	46: IF Laser_Marked THEN
			OP150_Laser_Start:=0;
			OP150b_Auto_Seq :=47;
		END_IF	
		
	47:	IF NOT OP150_Laser_Start AND Laser_Marked THEN
			OP150b_Auto_Seq :=50;
		ELSIF OP150_Laser_Failed THEN		//Laser_Mark_Delay.Q AND (OP150_Laser_Failed OR NOT OP150_Laser_Completed) THEN
			OP150_Laser_Start:=0;
			OP150b_Auto_Seq :=80;
		END_IF
		
	50: MOVER_CMP_STATUS[OP150B_LH_STN_MOVER][1]:=156;	
		OP150B_LH_STN_ENABLE:=0;
		IF MOVER_CMP_STATUS[OP150B_LH_STN_MOVER][1]=156 THEN
			STATION_DONE[OP150B_LH_STN_MOVER][OP150B_LH_XTS_POS_NO]			:= TRUE;
			OP150b_Auto_Seq :=30;
		END_IF		
	
	60: Rejection_Code:=Rejection_Codes_Function(Fixture_LH);
		OP150B_Text_OK:=0;
		OP150b_Auto_Seq :=61;
		
	61: Line_1						:= Rejection_Code;
		OP150_Lsr_String  			:= Line_1; 
		OP150_Lsr_Block_ID			:= 0;
		OP150_Lsr_Text_Change_Start := 1;
		OP150b_Auto_Seq :=62;
		
	62:IF OP150_Lsr_Text_Change_Complete THEN// NOT OP150_Lsr_Text_Change_Start THEN
			Txt_Changed:=0;
			OP150b_Auto_Seq :=66;
		END_IF	
		
	66:	OP150_Laser_Start := TRUE;
		IF OP150_Laser_Start THEN
			OP150b_Auto_Seq :=67;
		END_IF	
	
	67: IF Laser_Marked THEN
			OP150_Laser_Start:=0;
			OP150b_Auto_Seq :=68;
		END_IF	
		
	68: IF NOT OP150_Laser_Start AND Laser_Marked THEN
			OP150b_Auto_Seq :=69;
		ELSIF OP150_Laser_Failed THEN//Laser_Mark_Delay.Q AND (OP150_Laser_Failed OR NOT OP150_Laser_Completed) THEN
			OP150_Laser_Start:=0;
			OP150b_Auto_Seq :=80;
		END_IF	
		
	69: Job_Initialize:=1;
		IF OP150B_Text_OK THEN
			OP150b_Auto_Seq:=70;
		END_IF
		
	70: OP150B_LH_STN_ENABLE:=0;
		MOVER_CMP_STATUS[OP150B_LH_STN_MOVER][1]:=156;	
		IF MOVER_CMP_STATUS[OP150B_LH_STN_MOVER][1]=156 THEN
			STATION_DONE[OP150B_LH_STN_MOVER][OP150B_LH_XTS_POS_NO]			:= TRUE;
			OP150b_Auto_Seq :=30;
		END_IF	

    80: MOVER_CMP_STATUS[OP150B_LH_STN_MOVER][1]:=157;
		IF MOVER_CMP_STATUS[OP150B_LH_STN_MOVER][1]=157 THEN
			OP150B_LH_STN_ENABLE:=0;
			OP150B_RH_STN_ENABLE:=0;
			STATION_DONE[OP150B_LH_STN_MOVER][OP150B_LH_XTS_POS_NO]	:= TRUE;
			OP150b_Auto_Seq :=30;
		END_IF		
		
	100: IF OP150B_Text_OK THEN //NOT OP150_Lsr_Text_Change_Start THEN
			OP150_Laser_Start := TRUE;
			IF OP150_Laser_Start THEN
				OP150b_Auto_Seq :=106;
			END_IF	
		 END_IF	
		
	106:IF Laser_Marked THEN
			OP150_Laser_Start:=0;
			OP150b_Auto_Seq :=107;
		END_IF	
		
	107:IF NOT OP150_Laser_Start AND Laser_Marked THEN
			OP150b_Auto_Seq :=110;
		ELSIF OP150_Laser_Failed THEN//Laser_Mark_Delay.Q AND (OP150_Laser_Failed OR NOT OP150_Laser_Completed) THEN
			OP150_Laser_Start:=0;
			OP150b_Auto_Seq :=160;
		END_IF
		
	110: OP150B_RH_STN_ENABLE:=0;
		 MOVER_CMP_STATUS[OP150B_RH_STN_MOVER][2]:=156;	
		 IF MOVER_CMP_STATUS[OP150B_RH_STN_MOVER][2]=156 THEN
			STATION_DONE[OP150B_RH_STN_MOVER][OP150B_RH_XTS_POS_NO]			:= TRUE;
			OP150b_Auto_Seq :=30;
		 END_IF		

	140: Rejection_Code:=Rejection_Codes_Function(Fixture_RH);
		 OP150b_Auto_Seq :=141;
		
	141: Line_1						:= Rejection_Code;
		 OP150_Lsr_String  			:= Line_1; 
		 OP150_Lsr_Block_ID			:= 0;
		 OP150_Lsr_Text_Change_Start := 1;
		 OP150b_Auto_Seq :=142;
		 
	142: IF OP150_Lsr_Text_Change_Complete THEN //NOT OP150_Lsr_Text_Change_Start THEN			
			OP150b_Auto_Seq :=143;
		 END_IF	

	143:// Line_2			  			:= 'D7.89';
		 OP150_Lsr_String  			:= Line_2; 
		 OP150_Lsr_Block_ID			:= 65536;
		 OP150_Lsr_Text_Change_Start := 1;
		 OP150b_Auto_Seq :=144;
		 
	144: IF OP150_Lsr_Text_Change_Complete THEN // NOT OP150_Lsr_Text_Change_Start THEN
			OP150b_Auto_Seq :=145;
		 END_IF	
	 
	145: //Line_3			  			:='>PK25D<';
		 OP150_Lsr_String  			:= Line_3; 
		 OP150_Lsr_Block_ID			:= 131072;
		 OP150_Lsr_Text_Change_Start := 1;
		 OP150b_Auto_Seq :=146;
		 
	146: IF OP150_Lsr_Text_Change_Complete THEN // NOT OP150_Lsr_Text_Change_Start THEN
			OP150_Laser_Start := TRUE;
			IF OP150_Laser_Start THEN
				OP150b_Auto_Seq :=147;
			END_IF	
		 END_IF	
	
	147: OP150_Laser_Start:=0;
		IF NOT OP150_Laser_Start THEN
			OP150b_Auto_Seq :=148;
		END_IF		 
		 
	148: IF NOT OP150_Laser_Start AND Laser_Marked THEN
			OP150b_Auto_Seq :=150;
		 ELSIF Laser_Mark_Delay.Q AND OP150_Laser_Failed THEN // OR NOT OP150_Laser_Completed) THEN
			OP150_Laser_Start:=0;
			OP150b_Auto_Seq :=160;
		 END_IF	
		
	150: MOVER_CMP_STATUS[OP150B_RH_STN_MOVER][2]:=156;	
		 IF MOVER_CMP_STATUS[OP150B_RH_STN_MOVER][2]=156 THEN
			STATION_DONE[OP150B_RH_STN_MOVER][OP150B_RH_XTS_POS_NO]			:= TRUE;
			OP150B_RH_STN_ENABLE:=0;
			OP150b_Auto_Seq :=30;
		 END_IF	
		 
	160: OP150B_RH_STN_ENABLE:=0;
		 MOVER_CMP_STATUS[OP150B_RH_STN_MOVER][2]:=157;	
		 IF MOVER_CMP_STATUS[OP150B_RH_STN_MOVER][2]=157 THEN
			STATION_DONE[OP150B_RH_STN_MOVER][OP150B_RH_XTS_POS_NO]			:= TRUE;
			OP150b_Auto_Seq :=30;
		 END_IF		 
END_CASE

Laser_Mark_Delay(IN:= (OP150_HMI_Reset OR OP150_Laser_Start),PT:=T#1S);

IF Laser_Mark_Delay.Q THEN
	OP150_HMI_Reset:=0;
END_IF

//Timer(IN:=OP150b_Auto_Seq=46 OR OP150b_Auto_Seq=106 ,PT:=T#1500MS);
//Txt_Change_Tmr(IN:=OP150_Lsr_Text_Change_Start ,PT:=T#500MS);

//IF Txt_Change_Tmr.Q THEN
//	OP150_Lsr_Text_Change_Start:=0;
//END_IF

IF Dry_run THEN
	Fixture_LH	:=150;
	Fixture_RH  :=150;
ELSE	
   Fixture_LH:=MOVER_CMP_STATUS[OP150B_LH_STN_MOVER][1];
   Fixture_RH:=MOVER_CMP_STATUS[OP150B_RH_STN_MOVER][2];
END_IF


//***************************Job change according to model********************************************\\
IF OP150_Model='6.3' THEN
	OP150_Lsr_Job_ID:=131072;
ELSIF OP150_Model='7.89' THEN
	OP150_Lsr_Job_ID:=0;
END_IF

IF OP150_Model='6.3' AND OP150_Laser_FB.Curr_JOB_id=2 THEN
	OP150B_Job_OK:=1;
ELSIF OP150_Model='7.89' AND OP150_Laser_FB.Curr_JOB_id=0 THEN
	OP150B_Job_OK:=1;
ELSE
	OP150B_Job_OK:=0;
END_IF

CASE OP150b_Job_Change_Seq OF
	10: IF NOT OP150_B_ErrorActive THEN
		 	OP150b_Job_Change_Seq :=20;
		END_IF
		
	20: IF OP150_Lsr_Ready THEN
			OP150b_Job_Change_Seq :=30;
		END_IF
		
	25: IF OP150_Model='6.3' AND OP150_Laser_FB.Curr_JOB_id<>2 THEN
			OP150b_Job_Change_Seq :=30;
		ELSIF OP150_Model='7.89' AND OP150_Laser_FB.Curr_JOB_id<>0 THEN
			OP150b_Job_Change_Seq :=30; 	
		END_IF
		
	30: IF OP150_Laser_FB.Curr_JOB_id <> OP150_Lsr_Job_ID THEN
			OP150b_Job_Change_Seq :=40;
		END_IF
		
	40: OP150_Lsr_Job_Change_Start:=1;
		OP150b_Job_Change_Seq :=50;
	 		
	50: IF OP150_Lsr_Job_Change_Complete AND NOT OP150_Lsr_Job_Change_Start THEN
			OP150_Lsr_Job_Change_Start := 0;
			OP150b_Job_Change_Seq :=25;
		END_IF
	
END_CASE

//************************************ Lines change According to Model & Batch ********************\\

Temp_String:=CONCAT(WORD_TO_STRING(fbTime.systemTime.wDay),'-');//WORD_TO_STRING(fbTime.systemTime.wMonth));
Laser_Line1:=CONCAT(Temp_String,'Jan');

IF Line_1<>Laser_Line1 THEN
	Job_Initialize:=1;
END_IF

CASE OP150b_Text_Change_Seq OF 
	
	10: IF NOT OP150_B_ErrorActive THEN
		 	OP150b_Text_Change_Seq :=20;
		END_IF
		
	20: IF OP150_Lsr_Ready THEN
			OP150b_Text_Change_Seq :=30;
		END_IF

	30: IF Batch_Change OR Job_Initialize THEN
			OP150B_Text_OK:=0;
			OP150b_Text_Change_Seq :=40;
		END_IF
	
 	40:	 Line_1						 := Laser_Line1;
		 OP150_Lsr_String  			 := Line_1; 
		 OP150_Lsr_Block_ID			 := 0;
		 OP150b_Text_Change_Seq 	 :=41;
		 
	41:  OP150_Lsr_Text_Change_Start := 1;
		  OP150b_Text_Change_Seq 	 :=50;
		 
	50: IF OP150_Lsr_Text_Change_Complete THEN //NOT OP150_Lsr_Text_Change_Start THEN
			Txt_Changed:=0;
			OP150b_Text_Change_Seq 	 :=60;
		 END_IF	
		
	60:	OP150_Lsr_String  			:= Line_2; 
		OP150_Lsr_Block_ID			:= 65536;
		OP150_Lsr_Text_Change_Start := 1;
		OP150b_Text_Change_Seq 	 :=70;
		
	70:IF OP150_Lsr_Text_Change_Complete THEN //NOT OP150_Lsr_Text_Change_Start THEN
			Txt_Changed:=0;
			OP150b_Text_Change_Seq 	 :=80;
		END_IF	
	 
	80:	OP150_Lsr_String  			:= Line_3; 
		OP150_Lsr_Block_ID			:= 131072;
		OP150_Lsr_Text_Change_Start := 1;
		OP150b_Text_Change_Seq 	 :=90;

	90: IF OP150_Lsr_Text_Change_Complete THEN //NOT OP150_Lsr_Text_Change_Start THEN
			Txt_Changed:=0;
			OP150b_Text_Change_Seq 	 :=100;
		END_IF		
		
  100:	OP150B_Text_OK  :=1;
  		Batch_Change    :=0;
		Job_Initialize  :=0;
		OP150b_Text_Change_Seq 	 :=10;
END_CASE


//############################		OP150B STATION ENABLE CONDITION		##########################\\

	OP150B_LH_STN_MOVER					:= MOVER_POSITION[OP150B_LH_XTS_POS_NO];
	OP150B_RH_STN_MOVER					:= MOVER_POSITION[OP150B_RH_XTS_POS_NO];
	
IF AUTO_WITH_XTS THEN

//###########################		LH			##################################	

	IF 	OP150B_LH_STN_MOVER>0 THEN
	IF NOT(END_OF_CYCLE AND MOVER_CMP_STATUS[OP150B_LH_STN_MOVER][1]=5)THEN		
	OP150B_LH_STN_ENABLE:= MOVER_POS_RECHED[OP150B_LH_STN_MOVER] AND (MOVER_CMP_STATUS[OP150B_LH_STN_MOVER][1]<155);
	ELSE
	STATION_DONE[OP150B_LH_STN_MOVER][OP150B_LH_XTS_POS_NO]			:= TRUE;		
	END_IF
	ELSE
		OP150B_LH_STN_ENABLE	:= FALSE;
	END_IF
	
//###########################		RH			##################################	
	
	IF 	OP150B_RH_STN_MOVER>0 THEN
	IF NOT(END_OF_CYCLE AND MOVER_CMP_STATUS[OP150B_RH_STN_MOVER][2]=5)THEN		
		OP150B_RH_STN_ENABLE:= MOVER_POS_RECHED[OP150B_RH_STN_MOVER] AND (MOVER_CMP_STATUS[OP150B_RH_STN_MOVER][2]<155);
	ELSE
	STATION_DONE[OP150B_RH_STN_MOVER][OP150B_RH_XTS_POS_NO]			:= TRUE;		
	END_IF
	ELSE
		OP150B_RH_STN_ENABLE		:= FALSE;
	END_IF										
END_IF

END_PROGRAM

// ---- POUs/Programs/OP150/Rejection_Codes_Function.TcPOU
FUNCTION Rejection_Codes_Function : STRING
VAR_INPUT
	Fixture_Code	: INT;
END_VAR
VAR	

END_VAR

IF Fixture_Code = 0 OR Fixture_Code >151 THEN
	Rejection_Codes_Function:=' NA ';
END_IF
IF Fixture_Code = 21 THEN
	Rejection_Codes_Function:='  OP20';
END_IF
IF Fixture_Code = 31 THEN
	Rejection_Codes_Function:='  OP30';
END_IF
IF Fixture_Code = 41 THEN
	Rejection_Codes_Function:='  OP40';
END_IF
IF Fixture_Code = 51 THEN
	Rejection_Codes_Function:='  OP50';
END_IF
IF Fixture_Code = 61 THEN
	Rejection_Codes_Function:='  OP60';
END_IF
IF Fixture_Code = 71 THEN
	Rejection_Codes_Function:='  OP70';
END_IF
IF Fixture_Code = 81 THEN
	Rejection_Codes_Function:='  OP80';
END_IF
IF Fixture_Code = 91 THEN
	Rejection_Codes_Function:='  OP90';
END_IF
IF Fixture_Code = 111 THEN
	Rejection_Codes_Function:='  OP110';
END_IF
IF Fixture_Code = 121 THEN
	Rejection_Codes_Function:='  OP120';
END_IF
IF Fixture_Code = 131 THEN
	Rejection_Codes_Function:='  OP130';
END_IF
IF Fixture_Code = 141 THEN
	Rejection_Codes_Function:='  OP140';
END_IF
IF Fixture_Code = 151 THEN
	Rejection_Codes_Function:='  OP150-V';
END_IF

END_FUNCTION

// ---- POUs/Programs/OP150/OP150_Laser_FB.TcPOU
PROGRAM OP150_Laser_FB
VAR
	Laser_Marker : FB_Keyence_Laser_Steuerung;
	
	Genreal_Status AT %I*  : ST_KeyenceLaser_General_Status;
	IO_Status AT %I*  : ST_KeyenceLaser_IO_Status;
	Running_Status AT %I*  : ST_KeyenceLaser_Running_Status;	
	Function_Status_I AT %I*  : ST_KeyenceLaser_Function_Status_I;
	Control_Status AT %I*  : ST_KeyenceLaser_Control_Status;		
	Req_Complete_Status AT %I*  : ST_KeyenceLaser_General_Request_Completion_Status;
	Edit_Req_Comp_Status AT %I*  : ST_KeyenceLaser_Edit_Request_Completion_Status;
	Operation_Req_Comp_Status AT %I*  : ST_KeyenceLaser_Operation_Request_Completion_Status;
	Block_Edit_Req_Status AT %I*  : ST_KeyenceLaser_Block_Edit_Request_Completion_Status;
	Cmnd_Req_Status AT %I*  : ST_KeyenceLaser_Command_Request_Completion_Status;
	General_Req_Err_Status AT %I*  : ST_KeyenceLaser_General_Request_Error_Status;
	Edit_Request_Error_Statu AT %I*  : ST_KeyenceLaser_Edit_Request_Error_Status;
	Operation_Request_Error_Status AT %I*  : ST_KeyenceLaser_Operation_Request_Error_Status;
	Block_Edit_Request_Error_Status AT %I*  : ST_KeyenceLaser_Block_Edit_Request_Error_Status;
	Command_Request_Error AT %I*  : ST_KeyenceLaser_Command_Request_Error;
	
	General_Request AT %Q* : ST_KeyenceLaser_General_Request_I;	
	Edit_Request AT %Q* : ST_KeyenceLaser_Edit_Request;	
	Operating_Request AT %Q* : ST_KeyenceLaser_Operating_Request;	
	Block_Edit_Request AT %Q* : ST_KeyenceLaser_Block_Edit_Request;	
	Command_Request AT %Q* : ST_KeyenceLaser_Command_Request;	
	Function_Request AT %Q* : ST_KeyenceLaser_Function_Request_I;	
	General_Request_Completion_Clear AT %Q* : ST_KeyenceLaser_General_Request_Completion_Clear;	
	Edit_Request_Completion_Clear AT %Q* : ST_KeyenceLaser_Edit_Request_Completion_Clear;	
	Operating_Request_Completion_Clear AT %Q* : ST_KeyenceLaser_Operating_Request_Completion_Clear;	
	Block_Edit_Request_Completion_Clear AT %Q* : ST_KeyenceLaser_Block_Edit_Request_Completion_Clear;	
	Command_Request_Completion_Clear AT %Q* : ST_KeyenceLaser_Command_Request_Completion_Clear;	
	Parameter AT %Q* : UDINT;	
	User_Data AT %Q* : ARRAY [0..127] OF BYTE;	
	User_Data_Size AT %Q* : UINT;	
	Curr_JOB_id AT %I* : UINT;

	OP150B_STN_MOVER	: INT;

	OP150B_LH_STN_MOVER: INT;
	OP150B_RH_STN_MOVER: INT;
    OP150B_LH_STN_ENABLE: BOOL;
    OP150B_RH_STN_ENABLE: BOOL;	
	
	Complete_Delay : TON;
	tmp: BOOL;
	Error_Delay	: TON;


	Dry_run                 : BOOL;	

END_VAR

Laser_Marker(
	stGeneralStatus:= Genreal_Status, 
	stIOStatus:= IO_Status, 
	stRunningStatus:= Running_Status, 
	stFunctionStatus:= Function_Status_I, 
	stControlStatus:= Control_Status, 
	stGeneralRequestCompletionStatus:= Req_Complete_Status, 
	stEditRequestCompletionStatus:= Edit_Req_Comp_Status, 
	stOperationRequestCompletionStatus:= Operation_Req_Comp_Status, 
	stBlockEditRequestCompletionStatus:= Block_Edit_Req_Status, 
	stCommandRequestCompletionStatus:= Cmnd_Req_Status, 
	stGeneralRequestErrorStatus:= General_Req_Err_Status, 
	stEditRequestErrorStatus:= Edit_Request_Error_Statu, 
	stOperationRequestErrorStatus:= Operation_Request_Error_Status, 
	stBlockEditRequestErrorStatus:= Block_Edit_Request_Error_Status, 
	stCommandRequestError:= Command_Request_Error, 
	iErrorCode0:= , 
	iErrorCode1:= , 
	iCurrentProgramNumber:= Curr_JOB_id, 
	iCounterNumber:= , 
	iCounterValue:= , 
	iRankValue:= , 
	iISOIECTR29158Grade:= , 
	iTwoDCCodeResultUpdateCount:= , 
	iPrintCount:= , 
	iResultDataSizet:= , 
	aResultData:= , 
	bClear_Error:=HMI_Reset OR OP150_HMI_Reset , 
	bLasermarking_Start:= OP150_Laser_Start , 
	iProgramNr:= OP150_Lsr_Job_ID, 
	iBlockNr:= OP150_Lsr_Block_ID, 
	sText:= OP150_Lsr_String, 
	bSafetyOK:= OperationEnable, 
	bProgramChange_Start:= OP150_Lsr_Job_Change_Start, 
	bBlockChange_Start:= OP150_Lsr_Text_Change_Start, 
	stGeneralRequest=> General_Request, 
	stEditRequest=> Edit_Request, 
	stOperatingRequest=> Operating_Request, 
	stBlockEditRequest=> Block_Edit_Request, 
	stCommandRequest=> Command_Request, 
	stFunctionRequest=> Function_Request, 
	stGeneralRequestCompletionClear=> General_Request_Completion_Clear, 
	stEditRequestCompletionClear=>Edit_Request_Completion_Clear, 
	stOperatingRequestCompletionClear=> Operating_Request_Completion_Clear, 
	stBlockEditRequestCompletionClear=> Block_Edit_Request_Completion_Clear, 
	stCommandRequestCompletionClear=> Command_Request_Completion_Clear, 
	iparameter=> Parameter, 
	iUserDataSize=> User_Data_Size , 
	aUserData=> User_Data, 
	nTemp=> , 
	nTemp2ByteSwaped=> , 
	bError=>OP150_B_ErrorActive , 
	bLaserMarking_finished=>OP150_Laser_Completed , 
	bLaserMarking_failed=>OP150_Laser_Failed , 
	bProgChangeComplete=>OP150_Lsr_Job_Change_Complete , 
	bBlockChangeComplete=>OP150_Lsr_Text_Change_Complete , 
	bLaserReady=>OP150_Lsr_Ready , 
	bTXTSM_Laser_not_ready=> , 
	bTXTSM_Laser_Error=> );
	
Error_Delay(IN:= NOT OP150_Lsr_Ready,PT:=T#10S);
	
IF Error_Delay.Q THEN
	OP150_B_ErrorActive:=1;
END_IF

IF HMI_Reset OR OP150_HMI_Reset THEN
	OP150_B_ErrorActive:=0;
END_IF

END_PROGRAM

// ---- FB/Keyence_Laser/FB_Keyence_Laser_Steuerung.TcPOU
FUNCTION_BLOCK FB_Keyence_Laser_Steuerung
VAR_INPUT
	//Kommunikationsdaten Laser IN
	//stMachineStatus 						: ST_KeyenceLaser_Machine_Status;
	//stFunctionStatus 						: ST_KeyenceLaser_Function_Status;
	//stCompletionStatus 						: ST_KeyenceLaser_Completion_Status;
	//stErrorStatus							: ST_KeyenceLaser_ErrorStatus;
	//stErrorCodes							: ST_KeyenceLaser_Error_Codes;
	//stOperateParametere						: ST_KeyenceLaser_Operate_Parameter;
	//stTwoDCodeReadResult					: ST_KeyenceLaser_TwoD_Code_Read_Result;
	//Count_Result_Data_Count_Result_Data 	: DWORD;
	//Result_Data_128byte_Result_Data 		: STRING[128];
	
	
//communication laser IN	
	// machine status
	stGeneralStatus										: ST_KeyenceLaser_General_Status;
	stIOStatus											: ST_KeyenceLaser_IO_Status;
	stRunningStatus										: ST_KeyenceLaser_Running_Status;
	                                            
	// function status                          
	stFunctionStatus									: ST_KeyenceLaser_Function_Status_I;
	stControlStatus										: ST_KeyenceLaser_Control_Status;
	                                            
	// completion status                        
	stGeneralRequestCompletionStatus					: ST_KeyenceLaser_General_Request_Completion_Status;
	stEditRequestCompletionStatus						: ST_KeyenceLaser_Edit_Request_Completion_Status;
	stOperationRequestCompletionStatus					: ST_KeyenceLaser_Operation_Request_Completion_Status;
	stBlockEditRequestCompletionStatus					: ST_KeyenceLaser_Block_Edit_Request_Completion_Status;
	stCommandRequestCompletionStatus					: ST_KeyenceLaser_Command_Request_Completion_Status;
	                                            
	// Error Status                             
	stGeneralRequestErrorStatus							: ST_KeyenceLaser_General_Request_Error_Status;
	stEditRequestErrorStatus							: ST_KeyenceLaser_Edit_Request_Error_Status;
	stOperationRequestErrorStatus						: ST_KeyenceLaser_Operation_Request_Error_Status;
	stBlockEditRequestErrorStatus						: ST_KeyenceLaser_Block_Edit_Request_Error_Status;
	stCommandRequestError								: ST_KeyenceLaser_Command_Request_Error;
	                                            
	// error code                               
	iErrorCode0											: UINT;
	iErrorCode1											: UINT;
	                                            
	// operate parametere                       
	iCurrentProgramNumber								: UINT;
	iCounterNumber										: UINT;
	iCounterValue										: UDINT;
	iRankValue											: UINT;
	                                            
	// 2D code read result                      
	iISOIECTR29158Grade									: UINT;
	iTwoDCCodeResultUpdateCount							: UINT;
	                                            
	// count result data                        
	iPrintCount											: UDINT;
	                                            
	// result data 128byte                      
	iResultDataSizet									: UINT;
	aResultData											: ARRAY [0..127] OF BYTE;
	
	bLasermarking_Start 					: BOOL := 0;
//Allgemeine Signale in
	bClear_Error							: BOOL := 0;
	
	
	iProgramNr 								: UDINT;
	iBlockNr 								: UDINT;
	sText 									: STRING;
	bSafetyOK								: BOOL;
END_VAR
VAR_IN_OUT
	//Trigger_Laser start
	bProgramChange_Start 					: BOOL := 0;
	bBlockChange_Start 						: BOOL := 0;
END_VAR
VAR_OUTPUT
	//Kommunikationsdaten Laser OUT
	//stGeneralRequest						: ST_KeyenceLaser_General_Request;
	//stFunctionRequest						: ST_KeyenceLaser_Function_Request;
	//stRequestCompletionClear				: ST_KeyenceLaser_Request_Completion_Clear;
	//Request_Parameter_Request_No			: DWORD;
	//Request_Data_128byte_Request_Data 	: STRING[128];
	
//communication laser OUT	
	
	// general request
	stGeneralRequest									: ST_KeyenceLaser_General_Request_I;
	stEditRequest										: ST_KeyenceLaser_Edit_Request;
	stOperatingRequest									: ST_KeyenceLaser_Operating_Request;
	stBlockEditRequest									: ST_KeyenceLaser_Block_Edit_Request;
	stCommandRequest									: ST_KeyenceLaser_Command_Request;
	                                            
	// function request                         
	stFunctionRequest									: ST_KeyenceLaser_Function_Request_I;
	                                            
	//  request completion clear                
	stGeneralRequestCompletionClear						: ST_KeyenceLaser_General_Request_Completion_Clear;
	stEditRequestCompletionClear						: ST_KeyenceLaser_Edit_Request_Completion_Clear;
	stOperatingRequestCompletionClear					: ST_KeyenceLaser_Operating_Request_Completion_Clear;
	stBlockEditRequestCompletionClear					: ST_KeyenceLaser_Block_Edit_Request_Completion_Clear;
	stCommandRequestCompletionClear						: ST_KeyenceLaser_Command_Request_Completion_Clear;
	                                            
	// request parameter                        
	                                            
	iparameter											: UDINT;
	                                            
	// request data 128byte                     
	                                            
	iUserDataSize										: UINT;
	aUserData											: ARRAY [0..127] OF BYTE;
	nTemp									: WORD;
	nTemp2ByteSwaped						: WORD;

	
//Allgemeine Signale out
	bError									: BOOL := 0;
	bLaserMarking_finished					: BOOL := 0;
	bLaserMarking_failed 					: BOOL := 0;
	bProgChangeComplete 					: BOOL := 0;
	bBlockChangeComplete					: BOOL := 0;
	bLaserReady								: BOOL := 0;	
	bTXTSM_Laser_not_ready					: BOOL := 0;
	bTXTSM_Laser_Error						: BOOL := 0;
END_VAR

VAR
	RProgramChange							: R_Trig;
	TONProgramChange						: TON;
	RTONProgramChange						: R_Trig;
	RProgramChangeComplete					: R_Trig;
	TPProgramChangeComplete					: TP;
	FNrogramChangeComplete					: F_Trig;
	
	RBlockChange							: R_Trig;
	TONBlockChange							: TON;
	RTONBlockChange							: R_Trig;
	RBlockChangeComplete					: R_Trig;
	TPBlockChangeComplete					: TP;
	FNlockChangeComplete					: F_Trig;
	bHMFPReset								: BOOL;
	R_LaserStart							: R_TRIG;
END_VAR
VAR_TEMP
	bFPReset								: BOOL;
END_VAR

//#########################################################################
//ErrorReset###############################################################
//#########################################################################

bError := stGeneralStatus.Error_Status;
IF stGeneralStatus.Error_Status AND bClear_Error THEN
	stGeneralRequest.Error_Clear_Request := TRUE;
ELSE	
	stGeneralRequest.Error_Clear_Request := FALSE;
END_IF;



//#########################################################################
//Ausgabe Fehlermeldungen##################################################
//#########################################################################

bTXTSM_Laser_not_ready := NOT stGeneralStatus.Ready_Status AND bSafetyOK;
bTXTSM_Laser_Error	 := (stCommandRequestError.Command_Request_Error
						OR 	stOperationRequestErrorStatus.Counter_Down_Error
						OR stOperationRequestErrorStatus.Counter_Number_Change_Error
						OR stOperationRequestErrorStatus.Counter_Reset_Error
						OR stOperationRequestErrorStatus.Counter_Up_Error
						OR stOperationRequestErrorStatus.Counter_Value_Change_Error
						OR stOperationRequestErrorStatus.Program_Change_error
						OR stOperationRequestErrorStatus.Rank_Value_Change
						OR stGeneralRequestErrorStatus.Print_Error
						OR stGeneralRequestErrorStatus.Guide_Print_Error
						OR stGeneralRequestErrorStatus.Error_Clear_Error
						OR stGeneralRequestErrorStatus.Print_Stop_Error
						OR stGeneralRequestErrorStatus.TwoDC_Read_Error
						OR stEditRequestErrorStatus.Edit_Error
						OR stBlockEditRequestErrorStatus.Character_String_Change_Error
						OR stBlockEditRequestErrorStatus.Character_String_Printed_Read_Error
						OR stBlockEditRequestErrorStatus.Character_String_Setting_Read_Error
						OR stCommandRequestError.Command_Request_Error
						OR iErrorCode0 <> 0
						OR iErrorCode1 <> 0
						)
						AND bSafetyOK;

IF bTXTSM_Laser_not_ready OR bTXTSM_Laser_Error THEN
bLasermarking_finished := FALSE; //stCompletionStatus.Marking_Complete; //über Ablauf setzen!!!
bLaserMarking_failed := FALSE; //über Ablauf setzen!!!
END_IF

// cancel program change 

IF NOT bProgramChange_Start THEN
stOperatingRequest.Program_Change_Request:= FALSE;
bProgChangeComplete:= FALSE;
END_IF



// activate program change 

RProgramChange(CLK:= bProgramChange_Start 
				AND NOT bBlockChange_Start
				AND NOT stOperatingRequest.Program_Change_Request
				AND NOT	stBlockEditRequest.Character_String_Change_Request,
				Q=> );

IF RProgramChange.Q THEN
iparameter:= (iProgramNr);
END_IF

	
TONProgramChange(IN:= bProgramChange_Start
					AND NOT bBlockChange_Start
					AND NOT stOperatingRequest.Program_Change_Request
					AND NOT	stBlockEditRequest.Character_String_Change_Request, 
					PT:=T#10MS ,
					Q=> , ET=> );
					
RTONProgramChange(CLK:=TONProgramChange.Q , Q=> );		

IF RTONProgramChange.Q THEN
	stOperatingRequest.Program_Change_Request:= TRUE;
END_IF


// complete program change

RProgramChangeComplete(CLK:= stOperationRequestCompletionStatus.PROGRAM_Change_Complete , Q=> );

stOperatingRequestCompletionClear.Program_Change_Complete_Clear:= RProgramChangeComplete.Q AND stOperatingRequest.Program_Change_Request;


IF RProgramChangeComplete.Q AND stOperatingRequest.Program_Change_Request THEN
	stOperatingRequest.Program_Change_Request:= FALSE;
END_IF

TPProgramChangeComplete(IN:= RProgramChangeComplete.Q , PT:= T#1MS, Q=> , ET=> );

FNrogramChangeComplete(CLK:= TPProgramChangeComplete.Q, Q=> );

IF FNrogramChangeComplete.Q THEN
	bProgramChange_Start:= FALSE;
	bProgChangeComplete:=TRUE;
END_IF



// cancel block change 

IF NOT bBlockChange_Start THEN
	stBlockEditRequest.Character_String_Change_Request:= FALSE;
	bBlockChangeComplete:= FALSE;
END_IF

// activate block change 


RBlockChange(CLK:= bBlockChange_Start 
				AND NOT bProgramChange_Start
				AND NOT stOperatingRequest.Program_Change_Request
				AND NOT	stBlockEditRequest.Character_String_Change_Request,
				Q=> );

IF RBlockChange.Q THEN
iparameter:= iBlockNr;
nTemp := INT_TO_WORD(LEN(STR:=sText));
////Test 1
//nTemp2ByteSwaped := ROL(nTemp,8);
//MEMCPY(destAddr:=ADR(aUserData) , srcAddr:=ADR(nTemp2ByteSwaped) , n:=SIZEOF(nTemp) );
//MEMCPY(destAddr:=ADR(aUserData)+SIZEOF(nTemp) , srcAddr:=ADR(sText) , n:=SIZEOF(sText) );

iUserDataSize := WORD_TO_UINT(nTemp);
MEMCPY(destAddr:=ADR(aUserData), srcAddr:=ADR(sText) , n:=SIZEOF(sText) );

END_IF

	
TONBlockChange(IN:= bBlockChange_Start
					AND NOT bProgramChange_Start
					AND NOT stOperatingRequest.Program_Change_Request
					AND NOT	stBlockEditRequest.Character_String_Change_Request, 
					PT:=T#10MS ,
					Q=> , ET=> );
					
RTONBlockChange(CLK:=TONBlockChange.Q , Q=> );		

IF RTONBlockChange.Q THEN
	stBlockEditRequest.Character_String_Change_Request:= TRUE;
END_IF


// complete block change

RBlockChangeComplete(CLK:= stBlockEditRequestCompletionStatus.Character_String_Change_Complete , Q=> );

stBlockEditRequestCompletionClear.Character_String_Change_Complete_Clear:= RBlockChangeComplete.Q AND stBlockEditRequest.Character_String_Change_Request;


IF RBlockChangeComplete.Q AND stBlockEditRequest.Character_String_Change_Request THEN
	stBlockEditRequest.Character_String_Change_Request:= FALSE;
END_IF

TPBlockChangeComplete(IN:= RBlockChangeComplete.Q , PT:= T#1MS, Q=> , ET=> );

FNlockChangeComplete(CLK:= TPBlockChangeComplete.Q, Q=> );

IF FNlockChangeComplete.Q THEN
	bBlockChange_Start:= FALSE;
	bBlockChangeComplete:=TRUE;
END_IF



// start marking

stGeneralRequest.Print_Start_Request:= bLasermarking_Start;

R_LaserStart(CLK:=bLasermarking_Start);

IF R_LaserStart.Q THEN
	bLaserMarking_finished:= FALSE;
END_IF
// Laser ready

bLaserReady:= stGeneralStatus.Ready_Status;

// Output complete Marking

IF stGeneralRequestCompletionStatus.Marking_Complete_2 THEN
	bLasermarking_Start:= FALSE;
	bLaserMarking_finished:= TRUE;
END_IF	
IF stRunningStatus.Print_Busy_Status THEN
 	bLaserMarking_finished:= FALSE;
END_IF

// reset error
bFPReset:= bClear_Error AND NOT bHMFPReset;
bHMFPReset:= bClear_Error;

stGeneralRequest.Error_Clear_Request:=bFPReset;


// Marking failed
bLaserMarking_failed:= (bLasermarking_Start AND (bTXTSM_Laser_not_ready OR bTXTSM_Laser_Error)) OR stGeneralRequestErrorStatus.Print_Error;

END_FUNCTION_BLOCK

// ---- POUs/Programs/OP150/OP150_C.TcPOU
PROGRAM OP150_C
VAR
	OP150_Laser_Camera 			      : FB_Cognex_ProfiNET_1;
	OP150_C_Camera_Trigger		      : BOOL;
	OP150_C_Camera_Job_Change_start   : BOOL;
	OP150_C_Camera_Error			  : BOOL;
	OP150_C_Camera_Ready			  : BOOL;
	OP150_C_Camera_Online			  : BOOL;	
	
	OP150_C_Acquisition_Status   AT %I*  :Acquisition_Status;
	OP150_C_Inspection_Status    AT %I*  :Inspection_Status;	
	OP150_C_Acquisition_ID       AT %I*  :UINT;
	OP150_C_Inspection_ID   	 AT %I*  :UINT;
	OP150_C_Error_code      	 AT %I*  :UINT;
	OP150_C_Current_Job_ID  	 AT %I*  :UINT;
	OP150_C_Result_code     	 AT %I*  :UINT;
	OP150_C_Cam_Result      	 AT %I*  :ARRAY[0..63] OF BYTE;
	
	OP150_C_Acquisition_Control AT %Q*  : Acquisition_Control;
	OP150_C_Inspection_Control  AT %Q*  : Inspection_Control;
	OP150_C_Command_word		AT %Q*  : UINT;
	Error_status				      : STRING;
	OP150_C_Target_Job_ID				  : UINT;
	OP150_C_Loaded_Job_ID		    	  : UINT;
	OP150_C_Union                       : UNION_64Byte;
	OP150_C_Job_Change_Complete		  : BOOL;
	OP150_C_Job_Change_Error   		  : BOOL;
	OP150_C_Picture_Taken      		  : BOOL;
	B1 : BOOL;
	B2 : BOOL;
	
	OP150C_STN_MOVER	: INT;

	OP150C_LH_STN_MOVER : INT;
	OP150C_RH_STN_MOVER : INT;
    OP150C_LH_STN_ENABLE: BOOL;
    OP150C_RH_STN_ENABLE: BOOL;		
	Dry_run             : BOOL;
	Complete_Delay      : TON;
	Error_Delay	: TON;
	tmp: BOOL;
	
	OP150c_Auto_Seq: INT;
	Fixture_LH: INT;
	Fixture_RH: INT;
	Toggle_Pos : R_TRIG;
	Toggle_Neg : F_TRIG;
	LH_Cam_Completed : BOOL;	
	OP150C_LH_CMP_OK : BOOL;
	OP150C_RH_CMP_OK : BOOL;
END_VAR

Toggle_Pos(CLK:=OP150_C.OP150_C_Inspection_Status.Inspection_Completed);
Toggle_Neg(CLK:=OP150_C.OP150_C_Inspection_Status.Inspection_Completed);

IF Toggle_Pos.Q OR Toggle_Neg.Q THEN
	LH_Cam_Completed:=1;	
END_IF			

OP150_Laser_Camera(
	tTimeout:= , 
	sJob_Name:= , 
	camera_ready=> OP150_C_Camera_Ready,
	Camera_online=> OP150_C_Camera_Online,
	stCognex_record_status:=OP150_C_Acquisition_Status, 
	Acquisition_ID:=OP150_C_Acquisition_ID , 
	stCognex_Inspection_status:=OP150_C_Inspection_Status, 
	Error_Code:=OP150_C_Error_code , 
	wcommand_control_in:= OP150_C_Current_Job_ID, 
	aResults_64_Bytes:= OP150_C_Cam_Result, 
	number_of_inspections:=OP150_C_Inspection_ID , 
	iresult_code:= OP150_C_Result_code, 
	bTarget_job_ID:=OP150_C_Target_Job_ID , 
	Error_Status_message=> Error_status, 
	bError=> OP150_C_Camera_Error, 
	stCognex_record_control=>OP150_C_Acquisition_Control , 
	stCognex_inspection_control=>OP150_C_Inspection_Control , 
	wCommandControl_out=>OP150_C_Command_word , 
	aUser_data_64_Byte=> OP150_C_Union.aArrayOfByte, 
	bJob_loading_completed=>OP150_C_Job_Change_Complete, 
	bJob_load_failed=>OP150_C_Job_Change_Error , 
	bInspection_Result_IO=>  B1, 
	bInspection_Result_NIO=> B2, 
	bTXTSM_Error_Job_Change=> OP150_C_Job_Change_Error, 
	bPictureTakenComplete=> OP150_C_Picture_Taken, 
	Loaded_Job_ID=>OP150_C_Loaded_Job_ID	 , 
	bClear_Error:= HMI_Reset, 
	bJob_change_start:= OP150_C_Camera_Job_Change_start, 
	TXTSM_camera_not_online=>OP150_C_Camera_Error	 , 
	bTrigger_start:= OP150_C_Camera_Trigger );

	
IF HMI_Reset OR OP150_HMI_Reset THEN
	OP150_C_ErrorActive:=0;
END_IF	

Error_Delay(IN:= NOT OP150_C_Camera_Online,PT:=T#10S);
	
IF Error_Delay.Q THEN
	OP150_C_ErrorActive:=1;
END_IF	

IF OP150_C_ErrorActive OR NOT OperationEnable THEN
	OP150C_Auto_Seq:=10;
END_IF

CASE OP150C_Auto_Seq OF
	10: IF NOT OP150_C_ErrorActive THEN
		 	OP150C_Auto_Seq :=20;
		END_IF
		
	20: IF OP150_C_Camera_Online THEN
			OP150C_Auto_Seq :=30;
		END_IF
		
	30: IF OP150_C_Camera_Online THEN
			OP150C_RH_CMP_OK	:= FALSE;
			OP150C_LH_CMP_OK	:= FALSE;
			OP150C_Auto_Seq :=40;
		END_IF
	
	40: IF OP150C_LH_STN_ENABLE THEN
			IF Fixture_LH=156 THEN
				OP150C_Auto_Seq :=50;
			ELSE
				OP150C_Auto_Seq :=90;	
			END_IF
		ELSIF OP150C_RH_STN_ENABLE THEN
			IF  Fixture_RH=156 THEN
				OP150C_Auto_Seq :=100;
			ELSE
				OP150C_Auto_Seq :=90;	
			END_IF
		END_IF
		
	50: OP150_C_Camera_Trigger:=1;
		IF LH_Cam_Completed THEN
			OP150_C_Camera_Trigger:=0;
			OP150C_Auto_Seq :=60;
		END_IF	
	
	60: IF OP150_C_Cam_Result[0]=1  THEN
			OP150C_Auto_Seq :=70;	
		ELSIF OP150_C_Cam_Result[1]=1 THEN
			OP150C_Auto_Seq :=76;
		END_IF
			
	70:	OP150C_LH_CMP_OK	:= TRUE;
		OP150C_Auto_Seq :=75;
	
	75: MOVER_CMP_STATUS[OP150C_LH_STN_MOVER][1]:=158;
		IF MOVER_CMP_STATUS[OP150C_LH_STN_MOVER][1]=158 THEN
			OP150C_Auto_Seq :=80;
		END_IF

	76: MOVER_CMP_STATUS[OP150C_LH_STN_MOVER][1]	:=159;
		IF MOVER_CMP_STATUS[OP150C_LH_STN_MOVER][1] =159 THEN
			OP150C_Auto_Seq :=80;
		END_IF	
		
	80: OP150C_LH_STN_ENABLE:=0;
		LH_Cam_Completed:=0;
		STATION_DONE[OP150C_RH_STN_MOVER][OP150C_LH_XTS_POS_NO]	:= TRUE;
		OP150C_Auto_Seq :=30;
		
	90: OP150C_LH_STN_ENABLE:=0;
		OP150C_RH_STN_ENABLE:=0;
		STATION_DONE[OP150C_RH_STN_MOVER][OP150C_LH_XTS_POS_NO]	:= TRUE;
		OP150C_Auto_Seq :=30;	
		
	100:  OP150_C_Camera_Trigger:=1;
		IF LH_Cam_Completed THEN
			OP150_C_Camera_Trigger:=0;
			OP150C_Auto_Seq :=110;
		END_IF	
	
	110: IF OP150_C_Cam_Result[0]=1  THEN
			OP150C_Auto_Seq :=115;	
		ELSIF OP150_C_Cam_Result[1]=1 THEN
			OP150C_Auto_Seq :=126;
		END_IF
			
	115:OP150C_RH_CMP_OK:= TRUE;
		OP150C_Auto_Seq :=125;
		
	125: MOVER_CMP_STATUS[OP150C_RH_STN_MOVER][2]:=158;
		 IF MOVER_CMP_STATUS[OP150C_RH_STN_MOVER][2]=158 THEN
			OP150C_Auto_Seq :=130;
		 END_IF

	126:  MOVER_CMP_STATUS[OP150C_RH_STN_MOVER][2]:=159;
		 IF MOVER_CMP_STATUS[OP150C_RH_STN_MOVER][2]=159 THEN
			OP150C_Auto_Seq :=130;
		 END_IF	

	130: OP150C_RH_STN_ENABLE:=0;
		 LH_Cam_Completed:=0;
	 	 STATION_DONE[OP150C_RH_STN_MOVER][OP150C_RH_XTS_POS_NO]:= TRUE;
		 OP150C_Auto_Seq :=30;	
END_CASE

IF Dry_run THEN	
 Fixture_LH:=156;
 Fixture_RH:=156;
ELSE
 Fixture_LH :=MOVER_CMP_STATUS[OP150C_LH_STN_MOVER][1];
 Fixture_RH:= MOVER_CMP_STATUS[OP150C_RH_STN_MOVER][2];
END_IF

(*IF 	OP150A_LH_Start AND NOT OP150_C_ErrorActive AND OP150_C_Camera_Ready AND OP150_C_Camera_Online THEN
 	IF  MOVER_CMP_STATUS[OP150C_LH_STN_MOVER][1]=156 THEN	
		OP150_C_Camera_Trigger:=1;
		tmp:=1;
		IF OP150_C_Cam_Result[0]=1 AND Complete_Delay.Q THEN
			OP150_C_Camera_Trigger:=0;
			MOVER_CMP_STATUS[OP150C_LH_STN_MOVER][1]:=160;
			tmp:=1;
			IF Complete_Delay.Q AND MOVER_CMP_STATUS[OP150C_LH_STN_MOVER][1]=160 THEN
//				ALL_STATION_DONE.POSITION_DONE[OP150C_LH_XTS_POS_NO]:= TRUE;
				OP150C_LH_Start:=0;
			END_IF
		ELSIF OP150_C_Cam_Result[0]=2 AND Complete_Delay.Q THEN
			OP150_C_Camera_Trigger:=0;
			MOVER_CMP_STATUS[OP150C_LH_STN_MOVER][1]:=161;
			tmp:=1;
			IF Complete_Delay.Q AND MOVER_CMP_STATUS[OP150C_LH_STN_MOVER][1]=161 THEN
//				ALL_STATION_DONE.POSITION_DONE[OP150C_LH_XTS_POS_NO]:= TRUE;
				OP150C_LH_Start:=0;
			END_IF	
		END_IF
 	ELSIF MOVER_CMP_STATUS[OP150C_LH_STN_MOVER][1]<>156 THEN
		 	MOVER_CMP_STATUS[OP150C_LH_STN_MOVER][2]:=161;
//			ALL_STATION_DONE.POSITION_DONE[OP150C_LH_XTS_POS_NO]:= TRUE;
			OP150C_LH_Start:=0;
 	END_IF	
END_IF
	
IF 	OP150C_RH_Start AND NOT OP150_C_ErrorActive AND OP150_C_Camera_Ready AND OP150_C_Camera_Online THEN
 	IF  MOVER_CMP_STATUS[OP150C_RH_STN_MOVER][2]=156 THEN	
		OP150_C_Camera_Trigger:=1;
		tmp:=1;
		IF OP150_C_Cam_Result[0]=1 AND Complete_Delay.Q THEN
			OP150_C_Camera_Trigger:=0;
			MOVER_CMP_STATUS[OP150C_RH_STN_MOVER][2]:=160;
			tmp:=1;
			IF Complete_Delay.Q AND MOVER_CMP_STATUS[OP150C_RH_STN_MOVER][2]=160 THEN
//				ALL_STATION_DONE.POSITION_DONE[OP150C_RH_XTS_POS_NO]:= TRUE;
				OP150C_RH_Start:=0;
			END_IF
		ELSIF OP150_C_Cam_Result[0]=2 AND Complete_Delay.Q  THEN
			OP150_C_Camera_Trigger:=0;
			MOVER_CMP_STATUS[OP150C_RH_STN_MOVER][2]:=161;
			tmp:=1;
			IF Complete_Delay.Q AND MOVER_CMP_STATUS[OP150C_RH_STN_MOVER][2]=161 THEN
//				ALL_STATION_DONE.POSITION_DONE[OP150C_RH_XTS_POS_NO]:= TRUE;
				OP150C_RH_Start:=0;
			END_IF	
		END_IF
 	ELSIF MOVER_CMP_STATUS[OP150C_RH_STN_MOVER][2]<>156 THEN
		 	MOVER_CMP_STATUS[OP150C_RH_STN_MOVER][2]:=161;
//			ALL_STATION_DONE.POSITION_DONE[OP150C_RH_XTS_POS_NO]:= TRUE;
			OP150C_RH_Start:=0;
 	END_IF	
END_IF	
*)


//###########################################################################################################################################

	
OP150C_LH_STN_MOVER					:= MOVER_POSITION[OP150C_LH_XTS_POS_NO];
OP150C_RH_STN_MOVER					:= MOVER_POSITION[OP150C_RH_XTS_POS_NO];	
	
IF AUTO_WITH_XTS THEN
	IF 	OP150C_LH_STN_MOVER>0  THEN
		OP150C_LH_STN_ENABLE := MOVER_POS_RECHED[OP150C_LH_STN_MOVER] AND (MOVER_CMP_STATUS[OP150C_LH_STN_MOVER][1]>150);
	END_IF
	IF 	OP150C_RH_STN_MOVER>0  THEN	 
		OP150C_RH_STN_ENABLE := MOVER_POS_RECHED[OP150C_RH_STN_MOVER] AND (MOVER_CMP_STATUS[OP150C_RH_STN_MOVER][2]>150);
	END_IF	
END_IF

END_PROGRAM

// ---- POUs/Programs/XTS/MAIN_1.TcPOU
PROGRAM MAIN_1
VAR
	
// BOOL
	bInit							: BOOL;
	xtsReady						: BOOL;
	bStartMover1Detection			: BOOL;	
	bMover1DetectionComplete		: BOOL;
	bStartGrouping					: BOOL;
	bAllAxesReset					: BOOL;
	bAllAxesEnabled					: BOOL;
	bXtsReadyForSequence			: BOOL;
	bm1_staus_31					: BOOL;
	bm1_staus_32					: BOOL;	
	
// INT
	i								: UDINT;
	
// AXIS CONTROL
	mc_AddAxisToGroup				: ARRAY[1..nNumberOfMovers] OF MC_AddAxisToGroup;
	mc_Power						: ARRAY[1..nNumberOfMovers] OF MC_Power;
	mc_Reset						: ARRAY[1..nNumberOfMovers] OF MC_Reset;

// MC GROUP
	mcGroupEnable					: Mc_GroupEnable;
	mcGroupReset					: MC_GroupReset;

END_VAR

// Cyclic call of  fbXTSenvironment.
fbXTSEnvironment(bBusy=> , bDone=> , bError=> , ipResultMessage=> );

// Initialize fbXTSenvironment.
IF NOT bInit THEN
	IF fbXTSEnvironment.Init(TRUE) THEN
		fbXTSEnvironment.Init(FALSE);
		bInit :=TRUE;
	END_IF
	RETURN;
END_IF

// Check for all Position valid, is Teaching valid and movers found
IF fbXTSEnvironment.XpuTcIo(1).GetAreAllPositionsValid() AND
	fbXTSEnvironment.XpuTcIo(1).GetIsTeachingValid() 	 AND
	(fbXTSEnvironment.XpuTcIo(1).GetExpectedMoverCount() 	 =
	 fbXTSEnvironment.XpuTcIo(1).GetDetectedMoverCount() ) THEN
	 xtsReady	:=TRUE;
	 ELSE
	 	 xtsReady	:=FALSE;	 
	     RETURN;
END_IF

// Check for Mover 1 configuration.
IF fbXTSEnvironment.XpuTcIo(1).GetMoverIdDetectionMode() = MoverIdDetectionMode.Mover1 THEN
	IF bStartMover1Detection AND NOT fbXTSEnvironment.XpuTcIo(1).GetIsMoverIdDetectionActive()AND NOT fbXTSEnvironment.XpuTcIo(1).GetIsMoverIdDetectionValid 	()	THEN
		bStartMover1Detection	:=FALSE;
		fbXTSEnvironment.XpuTcIo(1).TriggerMoverIdDetection();		
	END_IF
	// Check for error in mover 1
	IF fbXTSEnvironment.XpuTcIo(1).GetIsMoverIdDetectionValid() THEN
		bMover1DetectionComplete	:=TRUE;
	ELSE
		bMover1DetectionComplete	:=FALSE;
		RETURN;	
	END_IF
END_IF

// CA Group Handling
(*IF nCAGroupState<> 50 THEN//AND Pulse_Block.Q5Hz THEN
	bStartGrouping		:= TRUE;
END_IF*)
IF bStartGrouping THEN nCAGroupState:=0; END_IF
CASE nCAGroupState OF  
		0:// Groupling of CA
		
		IF bStartGrouping THEN
			bStartGrouping := FALSE;
			nCAGroupState := 10;
		END_IF
		
		10: // Add axes in CA group
		FOR i:= 1 TO  nNumberOfMovers BY 1 DO	

		mc_AddAxisToGroup[i](
			AxesGroup:= CAGroup , 
			Axis:= Mover[i] ,
			Execute:= FALSE , 
			IdentInGroup:= udint_to_identingroup(i) , 
			Done=> , 
			Busy=> , 
			Error=> , 
			ErrorId=> );
		END_FOR
		nCAGroupState := 11;
		
		11://
		FOR i:= 1 TO  nNumberOfMovers BY 1 DO	

		mc_AddAxisToGroup[i](
			AxesGroup:= CAGroup , 
			Axis:= Mover[i] ,
			Execute:= TRUE , 
			IdentInGroup:= udint_to_identingroup(i) , 
			Done=> , 
			Busy=> , 
			Error=> , 
			ErrorId=> );
		END_FOR
		
		IF CAGroup.NcToPlc.Common.GroupAxesCount = nNumberOfMovers THEN
			nCAGroupState := 20;
		END_IF
		
		20:// Rest Movers false
		FOR i:= 1 TO  nNumberOfMovers BY 1 DO	
			mc_Reset[i](
				Axis:=Mover[i]  , 
				Execute:= FALSE, 
				Done=> , 
				Busy=> , 
				Error=> , 
				ErrorID=> );			
		END_FOR
			nCAGroupState := 21;
			
			21:// Rest Movers True
			bAllAxesReset:=TRUE;
				FOR i:= 1 TO  nNumberOfMovers  DO	
				mc_Reset[i](
				Axis:=Mover[i]  , 
				Execute:= TRUE, 
				Done=> , 
				Busy=> , 
				Error=> , 
				ErrorID=> );
				IF mc_Reset[i].Done THEN
				i:=i+1;
				END_IF
			END_FOR		
				bAllAxesReset:=bAllAxesReset AND NOT Mover[i].NcToPlc.StateDWord.31;
		IF bAllAxesReset THEN
			nCAGroupState := 30;
		END_IF
		
		30:// mover enable false
		FOR i:= 1 TO  nNumberOfMovers BY 1 DO	
		mc_Power[i](
			Axis:= Mover[i] , 
			Enable:= FALSE, 
			Enable_Positive:= TRUE , 
			Enable_Negative:= TRUE , 
			Override:=100 , 
			BufferMode:= , 
			Options:= , 
			Status=> , 
			Busy=> , 
			Active=> , 
			Error=> , 
			ErrorID=> );
			END_FOR
			nCAGroupState :=31;
			
			31:// mover enable
			i:=0;
		bAllAxesEnabled:=TRUE;
		FOR i:= 1 TO  nNumberOfMovers BY 1 DO	
		mc_Power[i](
			Axis:= Mover[i] , 
			Enable:= TRUE, 
			Enable_Positive:= TRUE , 
			Enable_Negative:= TRUE , 
			Override:=100 , 
			BufferMode:= , 
			Options:= , 
			Status=> , 
			Busy=> , 
			Active=> , 
			Error=> , 
			ErrorID=> );
			bAllAxesEnabled:= bAllAxesEnabled AND Mover[i].NcToPlc.StateDWord.0;

			END_FOR
			
			IF bAllAxesEnabled THEN 
					nCAGroupState :=35;
			END_IF
			
			35: // Disable group
			mcGroupReset(
				AxesGroup:= CAGroup, 
				Execute:= TRUE , 
				Done=> , 
				Busy=> , 
				Error=> , 
				ErrorId=> );
				IF mcGroupReset.Done THEN
					nCAGroupState :=36;
				END_IF
			
				36: // Disable False group
				mcGroupReset(
				AxesGroup:= CAGroup, 
				Execute:= FALSE , 
				Done=> , 
				Busy=> , 
				Error=> , 
				ErrorId=> );				
				nCAGroupState :=40;			
			
			40: //False Group
			mcGroupEnable(
				AxesGroup:=CAGroup , 
				Execute:= FALSE, 
				Done=> , 
				Busy=> , 
				Error=> , 
				ErrorId=> );
				nCAGroupState :=41;
			
			41: 	//Enable Group
			mcGroupEnable(
				AxesGroup:=CAGroup , 
				Execute:= TRUE, 
				Done=> , 
				Busy=> , 
				Error=> , 
				ErrorId=> );
			IF mcGroupEnable.Done THEN
				nCAGroupState :=50;
			END_IF
						
			50:	bXtsReadyForSequence :=TRUE;

			//55: PRG_XTS_Sequence(); 									//bXtsReadyForSequence :=TRUE;	
			
END_CASE

IF bXtsReadyForSequence THEN
	PRG_XTS_Sequence();
END_IF


bm1_staus_31:=Mover[1].NcToPlc.StateDWord.31;
bm1_staus_32:=Mover[2].NcToPlc.StateDWord.31;

END_PROGRAM

// ---- POUs/Programs/XTS/PRG_XTS_Sequence.TcPOU
PROGRAM PRG_XTS_Sequence
VAR	
	
// MOVER STATION POSITION AND VELOCITY ARRAY
	rStationPostion											: ARRAY [0..nNumberOfStations] OF LREAL ;
	lr_internal_vel_cmd										: LREAL :=100;
	rCalculatedPostion										: ARRAY[0..nNumberofMovers] OF ARRAY[0..nNumberOfStations]OF LREAL;
	rStationVelocity										: ARRAY[0..nNumberOfStations] OF LREAL ;
	XTS_STP_POS_2_D											: ARRAY[0..nNumberofMovers] OF ARRAY[0..nNumberOfStations]OF LREAL;
	STATION_POSS_DN											: ARRAY[0..nNumberofMovers] OF ARRAY[0..nNumberOfStations]OF BOOL;	
// MOVER FUNCTIONAL BLOCK
	FbMoverSequence											: ARRAY [0..nNumberofMovers] OF Fb_MoverSequence;
	bRunCmd													: BOOL; // MOVER START FOR AUTO LOGIC
	bStopCmd												: BOOL; //MOVER STOP AND ALLIGN AT ONE POSITION
	bPausCmd												: BOOL; // MOVER HAULT	
// INT,REAL
	XTS_POSITION_P_TOLERANCE								: LREAL		:=1;
	XTS_POSITION_N_TOLERANCE								: LREAL		:=-1;

//DECLERATION

	


// FOR LOOP INTEGER	
	X														: INT; // FOR LOOP
	Y														: INT; // FOR LOOP
	i														: INT; // FOR LOOP
	j														: INT; // FOR LOOP







 	
//FbMoverSequence_2Parallel_OP: ARRAY [1..nNumberofMovers] OF Fb_MoverSequence_2Parallel_OP;
//	bSt4Busy: BOOL;
//Fb_MoverSequence_time: Fb_MoverSequence;	
	TonWait_ST_PT: ARRAY [1..20] OF TIME := [TIME#800MS, TIME#900MS, TIME#800MS, TIME#850MS, TIME#800MS, TIME#850MS, TIME#800MS, TIME#850MS, TIME#800MS, TIME#850MS, TIME#900MS, TIME#1S100MS, TIME#1S200MS, TIME#1S500MS, TIME#400MS, TIME#700MS, TIME#700MS];
	bMover1_Cycle_Time_on: BOOL;
	bMover1_Cycle_Time_Timer: Ton;
	bMover1_Cycle_Time_on_Ftrig: F_TRIG;
	bMover1_Cycle_Time: TIME;

	MOVER_CNTINUE							: BOOL;
	OP10A_SAFE								: BOOL;
	OP10B_SAFE								: BOOL;	
	OP20_SAFE								: BOOL;
	OP30_SAFE								: BOOL;
	OP40_SAFE								: BOOL;	
	OP50_SAFE								: BOOL;	
	OP60_SAFE								: BOOL;	
	OP70_SAFE								: BOOL;	
	OP80_SAFE								: BOOL;	
	OP90_SAFE								: BOOL;
	OP110_SAFE								: BOOL;
	OP120_SAFE								: BOOL;
	OP130_SAFE								: BOOL;	
	OP140_SAFE								: BOOL;	
	OP150A_SAFE								: BOOL;
	OP150B_SAFE								: BOOL;
	OP160_SAFE								: BOOL;	
	done_check								: BOOL;
	rst_array_memory						: BOOL;	
	OP140_XTS_TARGET						: LREAL;
	XTS_LOGIC_CHECK: BOOL;
	PerMISSION: R_TRIG;
	ZERO_POS_MOVER: INT;
	ALL_MOVER_EMPTY: BOOL;
	END_OF_CYLE: R_TRIG;
END_VAR


VAR PERSISTENT

	MVR_POS_BYPAS_LOG_COUNT					: INT;
	COIL_1									: BOOL;
	COIL_2									: BOOL;	
	COIL_3									: BOOL;
	COIL_4									: BOOL;	
	COIL_5									: BOOL;	
END_VAR

FOR i :=1 TO nNumberOfMovers BY 1 DO
	FOR j:=1 TO nNumberOfStations BY 1 DO
			IF Mover[i].NcToPlc.ModuloSetPos > rStationPostion[j] THEN
			rCalculatedPostion[i][j] := (((Mover[i].NcToPlc.ModuloSetTurns +1 ) *9000) + rStationPostion[j]);
			ELSE
			rCalculatedPostion[i][j] := (((Mover[i].NcToPlc.ModuloSetTurns +0) *9000) + rStationPostion[j]);
			END_IF			
			rStationVelocity[j]:=lr_internal_vel_cmd;			
		IF (i MOD 2)<>0 THEN
			IF j=OP10A_XTS_POS_NO THEN
			STN_BYPASS_ARAAY[i][j]	:= NOT OP10B_BYPASS;
			ELSIF j=(OP10A_XTS_POS_NO+1) THEN
			STN_BYPASS_ARAAY[i][j]	:= OP10B_BYPASS;			
			ELSE
			STN_BYPASS_ARAAY[i][j]	:= STN_BYPASS_ARRAY_HMI[j];
			END_IF	
		ELSIF (i MOD 2)=0 THEN
			IF j=OP10B_XTS_POS_NO THEN
			STN_BYPASS_ARAAY[i][j]	:= NOT OP10A_BYPASS;
			ELSIF j=(OP10B_XTS_POS_NO+1) THEN
			STN_BYPASS_ARAAY[i][j]	:= OP10A_BYPASS;				
			ELSE
			STN_BYPASS_ARAAY[i][j]	:= STN_BYPASS_ARRAY_HMI[j];		
			END_IF
		END_IF
END_FOR
END_FOR

(*PerMISSION(CLK:=MOVER_POS_RECHED[OP130_STN_MOVER] , Q=> );
IF PerMISSION.Q THEN
	OP130_MVR_DN_PERMISSION		:= TRUE;
END_IF*)



IF (OP130_MVR_DN_PERMISSION) AND NOT COIL_2 AND NOT OP140_P3_BYPASS THEN
	XTS_STOP_POSITION[OP140_XTS_POS_NO]:= XTS_STOP_POSITION[OP140_P3_XTS_POS_NO];//7200.18;
	COIL_1							:= TRUE;
	OP130_MVR_DN_PERMISSION			:= FALSE;
	ELSIF OP140_P3_BYPASS THEN
	COIL_1							:= TRUE;		
END_IF

IF COIL_1 AND NOT OP130_MVR_DN_PERMISSION THEN
	COIL_2							:= TRUE;	
END_IF

IF (OP130_MVR_DN_PERMISSION) AND COIL_2 AND NOT COIL_3 AND NOT OP140_P2_BYPASS THEN
	XTS_STOP_POSITION[OP140_XTS_POS_NO]:= XTS_STOP_POSITION[OP140_P2_XTS_POS_NO];//7000.18;	
	COIL_3							:= TRUE;
	OP130_MVR_DN_PERMISSION			:= FALSE;
	ELSIF COIL_1 AND OP140_P2_BYPASS THEN
	COIL_3							:= TRUE;		
END_IF

IF COIL_3 AND NOT OP130_MVR_DN_PERMISSION THEN
	COIL_4							:= TRUE;
END_IF

IF OP130_MVR_DN_PERMISSION AND COIL_4 AND NOT OP140_P1_BYPASS THEN
	XTS_STOP_POSITION[OP140_XTS_POS_NO]:= XTS_STOP_POSITION[OP140_P1_XTS_POS_NO];//6799.26 ;
	COIL_5							:= TRUE;
	OP130_MVR_DN_PERMISSION			:= FALSE;
	ELSIF COIL_3 AND OP140_P1_BYPASS THEN
	COIL_5							:= TRUE;	
END_IF

IF COIL_5 AND NOT OP130_MVR_DN_PERMISSION THEN
	COIL_1							:= FALSE;
	COIL_2                          := FALSE;
	COIL_3                          := FALSE;
	COIL_4                          := FALSE;
	COIL_5                          := FALSE;
END_IF

(*IF XTS_LOGIC_CHECK	THEN
	FOR i:=0 TO nNumberOfStations BY 1 DO
	ALL_STATION_DONE.POSITION_DONE[i]:= TRUE;		
	END_FOR
	XTS_LOGIC_CHECK					:= FALSE;
	OP130_MVR_DN_PERMISSION			:= FALSE;
END_IF*)


FOR i :=1 TO nNumberOfMovers BY 1 DO
	FbMoverSequence[i](
										bRun:= bRunCmd, 
										bStop:=bStopCmd ,
										bPause:=bPausCmd, 
										rPosition:=rCalculatedPostion[i] , 
										rVelocity:=rStationVelocity,
										lrCaGap := 200 ,
										XTS_STP_POS	:= XTS_STP_POS_2_D[i],			
										ACTUAL_MOVER_MODULE_POS	:= Mover[i].NcToPlc.ModuloActPos,TonWait_PT:=TonWait_ST_PT ,
										MOVER_CONTINUE := MOVER_CNTINUE,
										POS_BYPASS := STN_BYPASS_ARAAY[i],
										MoverAxis:=Mover[i],
										STATIONDONE := STATION_DONE[i],
										nMoverSequence := MOVER_STP_NO[i],
									//	STATION_DONE := ALL_STATION_DONE,
										POSITION_DONE:= );									
										MOVER_POS_RECHED[i]	:= FbMoverSequence[i].POSITION_DONE;
END_FOR;


// Part out time of  1st mover
bMover1_Cycle_Time_Timer.IN := bMover1_Cycle_Time_on;
bMover1_Cycle_Time_Timer.PT:=T#120S;
bMover1_Cycle_Time_Timer();

//IF PRG_XTS_Sequence.FbMoverSequence[1].nMoverSequence = 10 THEN bMover1_Cycle_Time_on := TRUE; END_IF
//IF PRG_XTS_Sequence.FbMoverSequence[1].nMoverSequence = 175 THEN bMover1_Cycle_Time_on := FALSE; END_IF


bMover1_Cycle_Time_on_Ftrig(CLK:= bMover1_Cycle_Time_on, Q=> );

IF bMover1_Cycle_Time_on_Ftrig.Q THEN bMover1_Cycle_Time :=bMover1_Cycle_Time_Timer.et; END_IF

(*
FOR i :=1 TO nNumberOfMovers BY 1 DO
	FbMoverSequence_2Parallel_OP[i](
									bRun:=bRunCmd , 
									bStop:=bStopCmd , 
									rPosition:=rCalculatedPostion[i] , 
									rVelocity:=rStationVelocity , 
									lrCaGap:= 100, 
									bSt4Busy:= bSt4Busy, 
									MoverAxis:= Mover[i]);
END_FOR

*)
FOR X:=1 TO nNumberOfStations DO
	rStationPostion[X]:= XTS_STOP_POSITION[X];
END_FOR

FOR i:=1 TO nNumberofMovers BY 1 DO
 	FOR j:=1 TO nNumberOfStations BY 1 DO
		XTS_STP_POS_2_D[i][j]:= XTS_STOP_POSITION[j];
	END_FOR
END_FOR


FOR X:=1 TO nNumberofMovers DO
FOR Y:=1 TO nNumberOfStations DO
	     MOVER_POSITION[Y]:=0;
 
END_FOR
END_FOR

FOR X:=1 TO nNumberofMovers DO
FOR Y:=1 TO nNumberOfStations DO
	IF ((Mover[X].NcToPlc.ModuloActPos-rStationPostion[Y])<=XTS_POSITION_P_TOLERANCE AND (Mover[X].NcToPlc.ModuloActPos-rStationPostion[Y])>0) OR
	   ((Mover[X].NcToPlc.ModuloActPos-rStationPostion[Y])>XTS_POSITION_N_TOLERANCE AND (Mover[X].NcToPlc.ModuloActPos-rStationPostion[Y])<0 ) THEN
	     MOVER_POSITION[Y]:=X;
	END_IF  
END_FOR
END_FOR

(*FOR X:=1 TO nNumberofMovers DO
FOR Y:=1 TO nNumberOfStations DO
	IF ((Mover[X].NcToPlc.ModuloActPos-rStationPostion[Y])<=XTS_POSITION_P_TOLERANCE AND (Mover[X].NcToPlc.ModuloActPos-rStationPostion[Y])>0) OR
	   ((Mover[X].NcToPlc.ModuloActPos-rStationPostion[Y])>XTS_POSITION_N_TOLERANCE AND (Mover[X].NcToPlc.ModuloActPos-rStationPostion[Y])<0 ) THEN
	     MOVER_POSITION[Y]:=X;
	END_IF  
END_FOR
END_FOR
*)






//#########################				SAFETY		#####################################


	IF OP20_SAFE AND OP30_SAFE AND OP40_SAFE AND OP50_SAFE AND OP60_SAFE AND OP70_SAFE AND OP80_SAFE AND 
		OP90_SAFE AND OP110_SAFE AND OP130_SAFE AND OP140_SAFE THEN
			bPausCmd			:= FALSE;	
	ELSE	
			bPausCmd			:= FALSE;
	END_IF

	
IF NOT OP20_STN_ENABLE THEN
	OP20_SAFE			:=(OP20_SERVO_ON_SFE_WRK OR OP20_SERVO_ON_HOME);
END_IF

IF NOT OP30_STN_ENABLE THEN
	OP30_SAFE			:=(OP30_VERT_SERVO_ON_HOME OR OP30_VERT_SERVO_ON_SFE_WRK);
END_IF

IF NOT OP40_STN_ENABLE THEN
	OP40_SAFE			:=(OP40_SERVO_ON_SFE_WRK OR OP40_SERVO_ON_HOME); 
END_IF 

IF NOT OP50_STN_ENABLE THEN
	OP50_SAFE			:=(OP50_VERT_SERVO_ON_SFE_WRK OR OP50_VERT_SERVO_ON_HOME); 
END_IF

IF NOT OP60_STN_ENABLE THEN
	OP60_SAFE			:=(OP60_SERVO_ON_SFE_WRK OR OP60_SERVO_ON_HOME); 
END_IF

IF NOT OP70_STN_ENABLE THEN
	OP70_SAFE			:=(OP70_VERT_SERVO_ON_SFE_WRK OR OP70_VERT_SERVO_ON_HOME); 
END_IF

IF NOT OP80_STN_ENABLE THEN
	OP80_SAFE			:=(OP80_SERVO_ON_SFE_WRK OR OP80_SERVO_ON_HOME); 
END_IF

IF NOT OP90_STN_ENABLE THEN
	OP90_SAFE			:=(OP90_SRV_LH_VERT_CNTRL.Axis_In_Pos AND (OP90_SRV_LH_VRT_HME_FB OR OP90_SRV_LH_VRT_SPLCWRK_FB)) AND 
							(OP90_SRV_RH_VERT_CNTRL.Axis_In_Pos AND (OP90_SRV_RH_VRT_HME_FB OR OP90_SRV_RH_VRT_SPLCWRK_FB));(* AND 
							  (OP90_SUP_HORZP1_CYL.Sensor1 AND OP90_SUP_HORZP2_CYL.Sensor1); *)
END_IF

IF NOT OP110_STN_ENABLE THEN
	OP110_SAFE			:=(OP110_SERVO_ON_SFE_WRK OR OP110_SERVO_ON_HOME); 
END_IF

IF NOT OP130_STN_ENABLE THEN
	OP130_SAFE			:=OP130_Temp_Home_OK;
END_IF

//IF NOT OP140_STN_ENABLE THEN
//	OP140_SAFE			:=OP140_Temp_Home_Ok;
//END_IF

	ZERO_POS_MOVER									:= MOVER_POSITION[ZERO_POS_NO];	
	STATION_DONE[ZERO_POS_MOVER][ZERO_POS_NO]		:= done_check;
	
IF END_OF_CYCLE THEN
	ALL_MOVER_EMPTY			:= TRUE;
	FOR i:= 1 TO nNumberofMovers BY 1 DO 
		FOR j:= 1 TO 2 BY 1 DO 
		IF MOVER_CMP_STATUS[i][j]<>5 THEN
		ALL_MOVER_EMPTY			:= FALSE;	
		END_IF
END_FOR	
END_FOR
END_IF

END_OF_CYLE(CLK:=ALL_MOVER_EMPTY AND END_OF_CYCLE , Q=> );
IF END_OF_CYLE.Q THEN
	done_check			:= FALSE;
	END_OF_CYCLE		:= FALSE;
END_IF


IF rst_array_memory OR bRunCmd THEN
	FOR i :=1 TO nNumberOfMovers BY 1 DO
		FOR j :=1 TO 3 BY 1 DO
					MOVER_CMP_STATUS[i][j]:=0;
		END_FOR
END_FOR
END_IF

END_PROGRAM

// ---- POUs/Programs/XTS/Fb_MoverSequence.TcPOU
FUNCTION_BLOCK Fb_MoverSequence
VAR_INPUT
	bRun								:BOOL;
	bStop								:BOOL;
	bPause								:BOOL;
	rPosition							:ARRAY[0..nNumberOfStations] OF MC_lReal;
	rVelocity							:ARRAY[0..nNumberOfStations] OF MC_lReal;
	lrCaGap								:MC_LREAL := 100;
	TonWait_PT							:ARRAY[1..20] OF TIME;
	
	MOVER_CONTINUE						: BOOL;
	POS_BYPASS							: ARRAY[0..nNumberOfStations] OF BOOL;
	XTS_STP_POS							: ARRAY[0..nNumberOfStations] OF LREAL;
	ACTUAL_MOVER_MODULE_POS				: LREAL;
	
END_VAR
VAR_OUTPUT
	POSITION_DONE						: BOOL;
END_VAR
VAR
	R_TRIG_Run							: R_trig;
	R_TRIG_Stop							: R_trig;
	R_TRIG_continue						: R_trig;	
	mcMoveAbsoluteCA					: MC_MoveAbsoluteCA;
	bStopCommandTriggered 				: BOOL;
	TonWait_st							: ARRAY[1..20] OF tON;
	mc_moverhalt						: MC_HaltCA;
	i									: INT;

	
	axis_busy: BOOL;
END_VAR

VAR_IN_OUT
	MoverAxis							:Axis_Ref;
//	STATION_DONE						: STATION_DONE;
	STATIONDONE							: ARRAY [0..nNumberOfStations] OF BOOL;
	nMoverSequence						: INT;
END_VAR

VAR PERSISTENT

END_VAR

R_TRIG_Run(CLK:=bRun , Q=> );
R_TRIG_Stop(CLK:=bStop , Q=> );
R_TRIG_continue(CLK:=MOVER_CONTINUE , Q=> );

IF R_TRIG_Run.Q THEN
 	bStopCommandTriggered :=TRUE;
END_IF

IF R_TRIG_Run.Q THEN
		nMoverSequence:=0;
END_IF

	IF R_TRIG_continue.Q THEN
	IF (nMoverSequence-1)>0 THEN
		nMoverSequence :=nMoverSequence-1;
	ELSE
		nMoverSequence:=10;
	END_IF
	END_IF
IF NOT bPause THEN
	mc_moverhalt(
	Axis:= MoverAxis, 
	Execute:= FALSE , 
	Deceleration:= , 
	Jerk:= , 
	Gap:= , 
	Options:= , 
	Done=> , 
	Busy=> , 
	Active=> , 
	CommandAborted=> , 
	Error=> , 
	ErrorId=> );
CASE nMoverSequence OF 
	0: 
	IF R_TRIG_Run.Q THEN
		nMoverSequence :=10;
	END_IF

	10:
	IF POS_BYPASS[1] THEN
	nMoverSequence:=20;
	ELSE
	mcMoveAbsoluteCA(
	Axis:=MoverAxis , 
	Execute:= FALSE, 
	ContinuousUpdate:= TRUE, 
	Position:= rPosition[1], 
	Velocity:= rVelocity [1], 
	Acceleration:= , 
	Deceleration:= , 
	Jerk:= , 
	Gap:= lrCaGap, 
	BufferMode:= , 
	Direction:= , 
	Options:= , 
	Done=> , 
	Busy=> , 
	Active=> , 
	CommandAborted=> , 
	Error=> , 
	ErrorId=> );
	STATIONDONE[1]			:=FALSE;
	IF 	STATIONDONE[1]=FALSE THEN
	nMoverSequence :=11;
	END_IF
 	END_IF

	
	11:
	IF POS_BYPASS[1] THEN
	nMoverSequence:=20;
	ELSE  
	mcMoveAbsoluteCA(
	Axis:=MoverAxis , 
	Execute:= TRUE, 
	ContinuousUpdate:= TRUE, 
	Position:= rPosition[1], 
	Velocity:= rVelocity [1], 
	Acceleration:= , 
	Deceleration:= , 
	Jerk:= , 
	Gap:= lrCaGap, 
	BufferMode:= , 
	Direction:= , 
	Options:= , 
	Done=> , 
	Busy=> axis_busy, 
	Active=> , 
	CommandAborted=> , 
	Error=> , 
	ErrorId=> );
	
	IF mcMoveAbsoluteCA.Done AND STATIONDONE[1] THEN
		nMoverSequence 							:=20;
		STATIONDONE[1]			:=FALSE;
	END_IF
	END_IF
//	TonWait_st[1](IN:=FALSE , PT:=TonWait_PT[1] , Q=> , ET=> );
	15:
(*	TonWait_st[1](IN:=TRUE , PT:=TonWait_PT[1] , Q=> , ET=> );
	IF TonWait_st[1].Q THEN
		nMoverSequence :=20;
	END_IF *)
	

	20:
	IF POS_BYPASS[2] THEN
	nMoverSequence:=30;
	ELSE 
	mcMoveAbsoluteCA(
	Axis:=MoverAxis , 
	Execute:= FALSE, 
	ContinuousUpdate:= TRUE, 
	Position:= rPosition[2], 
	Velocity:= rVelocity [2], 
	Acceleration:= , 
	Deceleration:= , 
	Jerk:= , 
	Gap:= lrCaGap , 
	BufferMode:= , 
	Direction:= , 
	Options:= , 
	Done=> , 
	Busy=> , 
	Active=> , 
	CommandAborted=> , 
	Error=> , 
	ErrorId=> );
	STATIONDONE[2]			:=FALSE;
	IF 	STATIONDONE[2]=FALSE THEN
	nMoverSequence :=21;
	END_IF
	END_IF 

	
	21:
	IF POS_BYPASS[2] THEN
	nMoverSequence:=30;
	ELSE 
	mcMoveAbsoluteCA(
	Axis:=MoverAxis , 
	Execute:= TRUE, 
	ContinuousUpdate:= TRUE, 
	Position:= rPosition[2], 
	Velocity:= rVelocity [2], 
	Acceleration:= , 
	Deceleration:= , 
	Jerk:= , 
	Gap:= lrCaGap, 
	BufferMode:= , 
	Direction:= , 
	Options:= , 
	Done=> , 
	Busy=> , 
	Active=> , 
	CommandAborted=> , 
	Error=> , 
	ErrorId=> );
	
	IF mcMoveAbsoluteCA.Done AND STATIONDONE[2] THEN
		nMoverSequence 							:=30;
		STATIONDONE[2]			:=FALSE;
	END_IF
	END_IF 

//	TonWait_st[2](IN:=FALSE , PT:=TonWait_PT[2] , Q=> , ET=> );
	25:
(*	TonWait_st[2](IN:=TRUE , PT:=TonWait_PT[2] , Q=> , ET=> );
	IF TonWait_st[2].Q THEN
		nMoverSequence :=30;
	END_IF *)
	
	

	
	30:
	IF POS_BYPASS[3] THEN
	nMoverSequence:=40;
	ELSE  
	mcMoveAbsoluteCA(
	Axis:=MoverAxis , 
	Execute:= FALSE, 
	ContinuousUpdate:= TRUE, 
	Position:= rPosition[3], 
	Velocity:= rVelocity [3], 
	Acceleration:= , 
	Deceleration:= , 
	Jerk:= , 
	Gap:= lrCaGap, 
	BufferMode:= , 
	Direction:= , 
	Options:= , 
	Done=> , 
	Busy=> , 
	Active=> , 
	CommandAborted=> , 
	Error=> , 
	ErrorId=> );
	STATIONDONE[3]:= FALSE;
	IF STATIONDONE[3]= FALSE THEN
	nMoverSequence :=31;		
	END_IF
	END_IF
	
	31:
	IF POS_BYPASS[3] THEN
	nMoverSequence:=40;
	ELSE 
	mcMoveAbsoluteCA(
	Axis:=MoverAxis , 
	Execute:= TRUE, 
	ContinuousUpdate:= TRUE, 
	Position:= rPosition[3], 
	Velocity:= rVelocity [3], 
	Acceleration:= , 
	Deceleration:= , 
	Jerk:= , 
	Gap:= lrCaGap, 
	BufferMode:= , 
	Direction:= , 
	Options:= , 
	Done=> , 
	Busy=> , 
	Active=> , 
	CommandAborted=> , 
	Error=> , 
	ErrorId=> );
	
	IF mcMoveAbsoluteCA.Done AND STATIONDONE[3] THEN
		nMoverSequence :=40;
		STATIONDONE[3]			:=FALSE;
	END_IF
	END_IF
//	TonWait_st[3](IN:=FALSE , PT:=TonWait_PT[3] , Q=> , ET=> );
	
	35:
(*	TonWait_st[3](IN:=TRUE , PT:=TonWait_PT[3] , Q=> , ET=> );
	IF TonWait_st[3].Q THEN
		nMoverSequence :=40;
	END_IF*)
	
	
	40:
	IF POS_BYPASS[4] THEN
	nMoverSequence:=50;
	ELSE  
	mcMoveAbsoluteCA(
	Axis:=MoverAxis , 
	Execute:= FALSE, 
	ContinuousUpdate:= TRUE, 
	Position:= rPosition[4], 
	Velocity:= rVelocity [4], 
	Acceleration:= , 
	Deceleration:= , 
	Jerk:= , 
	Gap:= lrCaGap, 
	BufferMode:= , 
	Direction:= , 
	Options:= , 
	Done=> , 
	Busy=> , 
	Active=> , 
	CommandAborted=> , 
	Error=> , 
	ErrorId=> );
	STATIONDONE[4]:= FALSE;
	IF STATIONDONE[4]= FALSE THEN
	nMoverSequence :=41;		
	END_IF
	END_IF
	
	
	
	41:
	IF POS_BYPASS[4] THEN
	nMoverSequence:=50;
	ELSE 
	mcMoveAbsoluteCA(
	Axis:=MoverAxis , 
	Execute:= TRUE, 
	ContinuousUpdate:= TRUE, 
	Position:= rPosition[4], 
	Velocity:= rVelocity [4], 
	Acceleration:= , 
	Deceleration:= , 
	Jerk:= , 
	Gap:= lrCaGap , 
	BufferMode:= , 
	Direction:= , 
	Options:= , 
	Done=> , 
	Busy=> , 
	Active=> , 
	CommandAborted=> , 
	Error=> , 
	ErrorId=> );
	
	IF mcMoveAbsoluteCA.Done AND STATIONDONE[4] THEN
		nMoverSequence :=50;
		STATIONDONE[4]			:=FALSE;
	END_IF
	END_IF
//	TonWait_st[4](IN:=FALSE , PT:=TonWait_PT[4] , Q=> , ET=> );
	
	45:
(*	TonWait_st[4](IN:=TRUE , PT:=TonWait_PT[4] , Q=> , ET=> );
	IF TonWait_st[4].Q THEN
		nMoverSequence :=50;
	END_IF*)
	
	
	50:
	IF POS_BYPASS[5] THEN
	nMoverSequence:=60;
	ELSE 
	mcMoveAbsoluteCA(
	Axis:=MoverAxis , 
	Execute:= FALSE, 
	ContinuousUpdate:= TRUE, 
	Position:= rPosition[5], 
	Velocity:= rVelocity [5], 
	Acceleration:= , 
	Deceleration:= , 
	Jerk:= , 
	Gap:= lrCaGap , 
	BufferMode:= , 
	Direction:= , 
	Options:= , 
	Done=> , 
	Busy=> , 
	Active=> , 
	CommandAborted=> , 
	Error=> , 
	ErrorId=> );
	STATIONDONE[5]:= FALSE;
	IF STATIONDONE[5]= FALSE THEN
	nMoverSequence :=51;		
	END_IF
	END_IF
	
	51: 
	IF POS_BYPASS[5] THEN
	nMoverSequence:=60;
	ELSE 	
	mcMoveAbsoluteCA(
	Axis:=MoverAxis , 
	Execute:= TRUE, 
	ContinuousUpdate:= TRUE, 
	Position:= rPosition[5], 
	Velocity:= rVelocity [5], 
	Acceleration:= , 
	Deceleration:= , 
	Jerk:= , 
	Gap:= lrCaGap, 
	BufferMode:= , 
	Direction:= , 
	Options:= , 
	Done=> , 
	Busy=> , 
	Active=> , 
	CommandAborted=> , 
	Error=> , 
	ErrorId=> );
	
	IF mcMoveAbsoluteCA.Done AND STATIONDONE[5] THEN
		nMoverSequence :=60;
		STATIONDONE[5]			:=FALSE;
	END_IF
	END_IF
//	TonWait_st[5](IN:=FALSE , PT:=TonWait_PT[5] , Q=> , ET=> );
	
	55:
(*	TonWait_st[5](IN:=TRUE , PT:=TonWait_PT[5] , Q=> , ET=> );
	IF TonWait_st[5].Q THEN
		nMoverSequence :=60;
	END_IF*)
	
	
	60:
	IF POS_BYPASS[6] THEN
	nMoverSequence:=70;
	ELSE  
	mcMoveAbsoluteCA(
	Axis:=MoverAxis , 
	Execute:= FALSE, 
	ContinuousUpdate:= TRUE, 
	Position:= rPosition[6], 
	Velocity:= rVelocity [6], 
	Acceleration:= , 
	Deceleration:= , 
	Jerk:= , 
	Gap:= lrCaGap , 
	BufferMode:= , 
	Direction:= , 
	Options:= , 
	Done=> , 
	Busy=> , 
	Active=> , 
	CommandAborted=> , 
	Error=> , 
	ErrorId=> );
	STATIONDONE[6]:= FALSE;
	IF STATIONDONE[6]= FALSE THEN
	nMoverSequence :=61;
	END_IF
	END_IF

	61:
	IF POS_BYPASS[6] THEN
	nMoverSequence:=70;
	ELSE  
	mcMoveAbsoluteCA(
	Axis:=MoverAxis , 
	Execute:= TRUE, 
	ContinuousUpdate:= TRUE, 
	Position:= rPosition[6], 
	Velocity:= rVelocity [6], 
	Acceleration:= , 
	Deceleration:= , 
	Jerk:= , 
	Gap:= lrCaGap , 
	BufferMode:= , 
	Direction:= , 
	Options:= , 
	Done=> , 
	Busy=> , 
	Active=> , 
	CommandAborted=> , 
	Error=> , 
	ErrorId=> );
	
	IF mcMoveAbsoluteCA.Done AND STATIONDONE[6] THEN
		nMoverSequence :=70;
		STATIONDONE[6]			:=FALSE;
	END_IF
	END_IF	

//	TonWait_st[6](IN:=FALSE , PT:=TonWait_PT[6] , Q=> , ET=> );
	
	65:
(*	TonWait_st[6](IN:=TRUE , PT:=TonWait_PT[6] , Q=> , ET=> );
	IF TonWait_st[6].Q THEN
		nMoverSequence :=70;
	END_IF*)
	
	
	70:
	IF POS_BYPASS[7] THEN
	nMoverSequence:=80;
	ELSE 
	mcMoveAbsoluteCA(
	Axis:=MoverAxis , 
	Execute:= FALSE, 
	ContinuousUpdate:= TRUE, 
	Position:= rPosition[7], 
	Velocity:= rVelocity [7], 
	Acceleration:= , 
	Deceleration:= , 
	Jerk:= , 
	Gap:= lrCaGap , 
	BufferMode:= , 
	Direction:= , 
	Options:= , 
	Done=> , 
	Busy=> , 
	Active=> , 
	CommandAborted=> , 
	Error=> , 
	ErrorId=> );
	STATIONDONE[7]			:=FALSE;
	IF STATIONDONE[7]=FALSE THEN
	nMoverSequence :=71;
	END_IF
	END_IF
	
	71:
	IF POS_BYPASS[7] THEN
	nMoverSequence:=80;
	ELSE 
	mcMoveAbsoluteCA(
	Axis:=MoverAxis , 
	Execute:= TRUE, 
	ContinuousUpdate:= TRUE, 
	Position:= rPosition[7], 
	Velocity:= rVelocity [7], 
	Acceleration:= , 
	Deceleration:= , 
	Jerk:= , 
	Gap:= lrCaGap , 
	BufferMode:= , 
	Direction:= , 
	Options:= , 
	Done=> , 
	Busy=> , 
	Active=> , 
	CommandAborted=> , 
	Error=> , 
	ErrorId=> );
	
	IF mcMoveAbsoluteCA.Done AND STATIONDONE[7] THEN
		nMoverSequence :=80;
		STATIONDONE[7]			:=FALSE;
	END_IF
	END_IF
//	TonWait_st[7](IN:=FALSE , PT:=TonWait_PT[7] , Q=> , ET=> );
	
	75:
(*	TonWait_st[7](IN:=TRUE , PT:=TonWait_PT[7] , Q=> , ET=> );
	IF TonWait_st[7].Q THEN
		nMoverSequence :=80;
	END_IF*)
	
	
	80:
	IF POS_BYPASS[8] THEN
	nMoverSequence:=90;
	ELSE 
	mcMoveAbsoluteCA(
	Axis:=MoverAxis , 
	Execute:= FALSE, 
	ContinuousUpdate:= TRUE, 
	Position:= rPosition[8], 
	Velocity:= rVelocity [8], 
	Acceleration:= , 
	Deceleration:= , 
	Jerk:= , 
	Gap:= lrCaGap , 
	BufferMode:= , 
	Direction:= , 
	Options:= , 
	Done=> , 
	Busy=> , 
	Active=> , 
	CommandAborted=> , 
	Error=> , 
	ErrorId=> );
	STATIONDONE[8]:= FALSE;
	IF STATIONDONE[8]= FALSE THEN
	nMoverSequence :=81;
	END_IF
	END_IF
	
	81:
	IF POS_BYPASS[8] THEN
	nMoverSequence:=90;
	ELSE 
	mcMoveAbsoluteCA(
	Axis:=MoverAxis , 
	Execute:= TRUE, 
	ContinuousUpdate:= TRUE, 
	Position:= rPosition[8], 
	Velocity:= rVelocity [8], 
	Acceleration:= , 
	Deceleration:= , 
	Jerk:= , 
	Gap:= lrCaGap, 
	BufferMode:= , 
	Direction:= , 
	Options:= , 
	Done=> , 
	Busy=> , 
	Active=> , 
	CommandAborted=> , 
	Error=> , 
	ErrorId=> );
	
	IF mcMoveAbsoluteCA.Done AND STATIONDONE[8] THEN
		nMoverSequence :=90;
		STATIONDONE[8]			:=FALSE;
	END_IF
	END_IF
//	TonWait_st[8](IN:=FALSE , PT:=TonWait_PT[8] , Q=> , ET=> );
	
	85:
(*	TonWait_st[8](IN:=TRUE , PT:=TonWait_PT[8] , Q=> , ET=> );
	IF TonWait_st[8].Q THEN
		nMoverSequence :=90;
	END_IF*)
	
	
	90:
	IF POS_BYPASS[9] THEN
	nMoverSequence:=100;
	ELSE 
	mcMoveAbsoluteCA(
	Axis:=MoverAxis , 
	Execute:= FALSE, 
	ContinuousUpdate:= TRUE, 
	Position:= rPosition[9], 
	Velocity:= rVelocity [9], 
	Acceleration:= , 
	Deceleration:= , 
	Jerk:= , 
	Gap:= lrCaGap , 
	BufferMode:= , 
	Direction:= , 
	Options:= , 
	Done=> , 
	Busy=> , 
	Active=> , 
	CommandAborted=> , 
	Error=> , 
	ErrorId=> );
	STATIONDONE[9]:= FALSE;
	IF STATIONDONE[9]= FALSE THEN
	nMoverSequence :=91;
	END_IF
	END_IF
	
	91:
	IF POS_BYPASS[9] THEN
	nMoverSequence:=100;
	ELSE  
	mcMoveAbsoluteCA(
	Axis:=MoverAxis , 
	Execute:= TRUE, 
	ContinuousUpdate:= TRUE, 
	Position:= rPosition[9], 
	Velocity:= rVelocity [9], 
	Acceleration:= , 
	Deceleration:= , 
	Jerk:= , 
	Gap:= lrCaGap , 
	BufferMode:= , 
	Direction:= , 
	Options:= , 
	Done=> , 
	Busy=> , 
	Active=> , 
	CommandAborted=> , 
	Error=> , 
	ErrorId=> );
	
	IF mcMoveAbsoluteCA.Done AND STATIONDONE[9] THEN
		nMoverSequence :=100;
		STATIONDONE[9]			:=FALSE;
	END_IF
	END_IF
//	TonWait_st[9](IN:=FALSE , PT:=TonWait_PT[9] , Q=> , ET=> );
	
	95:
(*	TonWait_st[9](IN:=TRUE , PT:=TonWait_PT[9] , Q=> , ET=> );
	IF TonWait_st[9].Q THEN
		nMoverSequence :=100;
	END_IF *)
	
	
	100:
	IF POS_BYPASS[10] THEN
	nMoverSequence:=110;
	ELSE
	mcMoveAbsoluteCA(
	Axis:=MoverAxis , 
	Execute:= FALSE, 
	ContinuousUpdate:= TRUE, 
	Position:= rPosition[10], 
	Velocity:= rVelocity [10], 
	Acceleration:= , 
	Deceleration:= , 
	Jerk:= , 
	Gap:= lrCaGap, 
	BufferMode:= , 
	Direction:= , 
	Options:= , 
	Done=> , 
	Busy=> , 
	Active=> , 
	CommandAborted=> , 
	Error=> , 
	ErrorId=> );
	STATIONDONE[10]			:=FALSE;
	IF STATIONDONE[10]= FALSE THEN
	nMoverSequence :=101;
	END_IF
	END_IF
	
	101:
	IF POS_BYPASS[10] THEN
	nMoverSequence:=110;
	ELSE 
	mcMoveAbsoluteCA(
	Axis:=MoverAxis , 
	Execute:= TRUE, 
	ContinuousUpdate:= TRUE, 
	Position:= rPosition[10], 
	Velocity:= rVelocity [10], 
	Acceleration:= , 
	Deceleration:= , 
	Jerk:= , 
	Gap:= lrCaGap , 
	BufferMode:= , 
	Direction:= , 
	Options:= , 
	Done=> , 
	Busy=> , 
	Active=> , 
	CommandAborted=> , 
	Error=> , 
	ErrorId=> );
	
	IF mcMoveAbsoluteCA.Done AND STATIONDONE[10] THEN
		nMoverSequence :=110;
		STATIONDONE[10]			:=FALSE;
	END_IF
	END_IF
//	TonWait_st[10](IN:=FALSE , PT:=TonWait_PT[10] , Q=> , ET=> );
	
	105:
(*	TonWait_st[10](IN:=TRUE , PT:=TonWait_PT[10] , Q=> , ET=> );
	IF TonWait_st[10].Q THEN
		nMoverSequence :=110;
	END_IF*)
	
	
	110:
	IF POS_BYPASS[11] THEN
	nMoverSequence:=120;
	ELSE 
	mcMoveAbsoluteCA(
	Axis:=MoverAxis , 
	Execute:= FALSE, 
	ContinuousUpdate:= TRUE, 
	Position:= rPosition[11], 
	Velocity:= rVelocity [11], 
	Acceleration:= , 
	Deceleration:= , 
	Jerk:= , 
	Gap:= lrCaGap , 
	BufferMode:= , 
	Direction:= , 
	Options:= , 
	Done=> , 
	Busy=> , 
	Active=> , 
	CommandAborted=> , 
	Error=> , 
	ErrorId=> );
	STATIONDONE[11]			:=FALSE;
	IF STATIONDONE[11]=FALSE THEN
	nMoverSequence :=111;
	END_IF
	END_IF
	
	111:
	IF POS_BYPASS[11] THEN
	nMoverSequence:=120;
	ELSE  
	mcMoveAbsoluteCA(
	Axis:=MoverAxis , 
	Execute:= TRUE, 
	ContinuousUpdate:= TRUE, 
	Position:= rPosition[11], 
	Velocity:= rVelocity [11], 
	Acceleration:= , 
	Deceleration:= , 
	Jerk:= , 
	Gap:= lrCaGap, 
	BufferMode:= , 
	Direction:= , 
	Options:= , 
	Done=> , 
	Busy=> , 
	Active=> , 
	CommandAborted=> , 
	Error=> , 
	ErrorId=> );
	
	IF mcMoveAbsoluteCA.Done AND STATIONDONE[11] THEN
		nMoverSequence :=120;
		STATIONDONE[11]			:=FALSE;
	END_IF
	END_IF
//	TonWait_st[11](IN:=FALSE , PT:=TonWait_PT[11] , Q=> , ET=> );
	
	115:
(*	TonWait_st[11](IN:=TRUE , PT:=TonWait_PT[11] , Q=> , ET=> );
	IF TonWait_st[11].Q THEN
		nMoverSequence :=120;
	END_IF*)
	
	
	120:
	IF POS_BYPASS[12] THEN
	nMoverSequence:=130;
	ELSE  
	mcMoveAbsoluteCA(
	Axis:=MoverAxis , 
	Execute:= FALSE, 
	ContinuousUpdate:= TRUE, 
	Position:= rPosition[12], 
	Velocity:= rVelocity [12], 
	Acceleration:= , 
	Deceleration:= , 
	Jerk:= , 
	Gap:= lrCaGap , 
	BufferMode:= , 
	Direction:= , 
	Options:= , 
	Done=> , 
	Busy=> , 
	Active=> , 
	CommandAborted=> , 
	Error=> , 
	ErrorId=> );
		STATIONDONE[12]			:=FALSE;	
	IF STATIONDONE[12]=FALSE THEN
	nMoverSequence :=121;
	END_IF
	END_IF
	
	121:
	IF POS_BYPASS[12] THEN
	nMoverSequence:=130;
	ELSE 
	mcMoveAbsoluteCA(
	Axis:=MoverAxis , 
	Execute:= TRUE, 
	ContinuousUpdate:= TRUE, 
	Position:= rPosition[12], 
	Velocity:= rVelocity [12], 
	Acceleration:= , 
	Deceleration:= , 
	Jerk:= , 
	Gap:= lrCaGap, 
	BufferMode:= , 
	Direction:= , 
	Options:= , 
	Done=> , 
	Busy=> , 
	Active=> , 
	CommandAborted=> , 
	Error=> , 
	ErrorId=> );
	
	IF mcMoveAbsoluteCA.Done AND STATIONDONE[12] THEN
		nMoverSequence :=130;
		STATIONDONE[12]			:=FALSE;
	END_IF
	END_IF
//	TonWait_st[12](IN:=FALSE , PT:=TonWait_PT[12] , Q=> , ET=> );
	
	125:
(*	TonWait_st[12](IN:=TRUE , PT:=TonWait_PT[12] , Q=> , ET=> );
	IF TonWait_st[12].Q THEN
		nMoverSequence :=130;
	END_IF*)
	
	130:
	IF POS_BYPASS[13] THEN
	nMoverSequence:=140;
	ELSE 
	mcMoveAbsoluteCA(
	Axis:=MoverAxis , 
	Execute:= FALSE, 
	ContinuousUpdate:= TRUE, 
	Position:= rPosition[13], 
	Velocity:= rVelocity [13], 
	Acceleration:= , 
	Deceleration:= , 
	Jerk:= , 
	Gap:= lrCaGap, 
	BufferMode:= , 
	Direction:= , 
	Options:= , 
	Done=> , 
	Busy=> , 
	Active=> , 
	CommandAborted=> , 
	Error=> , 
	ErrorId=> );
	STATIONDONE[13]:=FALSE;
	IF STATIONDONE[13]=FALSE THEN
	nMoverSequence :=131;
	END_IF
	END_IF
	131:
	IF POS_BYPASS[13] THEN
	nMoverSequence:=140;
	ELSE 
	mcMoveAbsoluteCA(
	Axis:=MoverAxis , 
	Execute:= TRUE, 
	ContinuousUpdate:= TRUE, 
	Position:= rPosition[13], 
	Velocity:= rVelocity [13], 
	Acceleration:= , 
	Deceleration:= , 
	Jerk:= , 
	Gap:= lrCaGap , 
	BufferMode:= , 
	Direction:= , 
	Options:= , 
	Done=> , 
	Busy=> , 
	Active=> , 
	CommandAborted=> , 
	Error=> , 
	ErrorId=> );
	
	IF mcMoveAbsoluteCA.Done AND STATIONDONE[13] THEN
		nMoverSequence :=140;
		STATIONDONE[13]			:=FALSE;
	END_IF
	END_IF
//	TonWait_st[13](IN:=FALSE , PT:=TonWait_PT[13] , Q=> , ET=> );
	
	135:
(*	TonWait_st[13](IN:=TRUE , PT:=TonWait_PT[13] , Q=> , ET=> );
	IF TonWait_st[13].Q THEN
		nMoverSequence :=140;
	END_IF*)
	
	
	140:
	IF POS_BYPASS[14] THEN
	nMoverSequence:=150;
	ELSE  
	mcMoveAbsoluteCA(
	Axis:=MoverAxis , 
	Execute:= FALSE, 
	ContinuousUpdate:= TRUE, 
	Position:= rPosition[14], 
	Velocity:= rVelocity [14], 
	Acceleration:= , 
	Deceleration:= , 
	Jerk:= , 
	Gap:= lrCaGap, 
	BufferMode:= , 
	Direction:= , 
	Options:= , 
	Done=> , 
	Busy=> , 
	Active=> , 
	CommandAborted=> , 
	Error=> , 
	ErrorId=> );
	STATIONDONE[14]			:=FALSE;
	IF STATIONDONE[14]=FALSE THEN
	nMoverSequence :=141;
	END_IF
	END_IF
	141:
	IF POS_BYPASS[14] THEN
	nMoverSequence:=150;
	ELSE  
	mcMoveAbsoluteCA(
	Axis:=MoverAxis , 
	Execute:= TRUE, 
	ContinuousUpdate:= TRUE, 
	Position:= rPosition[14], 
	Velocity:= rVelocity [14], 
	Acceleration:= , 
	Deceleration:= , 
	Jerk:= , 
	Gap:= lrCaGap, 
	BufferMode:= , 
	Direction:= , 
	Options:= , 
	Done=> , 
	Busy=> , 
	Active=> , 
	CommandAborted=> , 
	Error=> , 
	ErrorId=> );
	
	IF mcMoveAbsoluteCA.Done AND STATIONDONE[14] THEN
		nMoverSequence :=150;
		STATIONDONE[14]			:=FALSE;
	END_IF
	END_IF
//	TonWait_st[14](IN:=FALSE , PT:=TonWait_PT[14] , Q=> , ET=> );
	
	145:
(*	TonWait_st[14](IN:=TRUE , PT:=TonWait_PT[14] , Q=> , ET=> );
	IF TonWait_st[14].Q THEN
		nMoverSequence :=150;
	END_IF*)
	
	
	150: 
	IF POS_BYPASS[15] THEN
	nMoverSequence:=160;
	ELSE 
	mcMoveAbsoluteCA(
	Axis:=MoverAxis , 
	Execute:= FALSE, 
	ContinuousUpdate:= TRUE, 
	Position:= rPosition[15], 
	Velocity:= rVelocity [15], 
	Acceleration:= , 
	Deceleration:= , 
	Jerk:= , 
	Gap:= lrCaGap, 
	BufferMode:= , 
	Direction:= , 
	Options:= , 
	Done=> , 
	Busy=> , 
	Active=> , 
	CommandAborted=> , 
	Error=> , 
	ErrorId=> );
	STATIONDONE[15]			:=FALSE;
	IF STATIONDONE[15]=FALSE THEN
	nMoverSequence :=151;
	END_IF
	END_IF
	
	151:
	IF POS_BYPASS[15] THEN
	nMoverSequence:=160;
	ELSE 
	mcMoveAbsoluteCA(
	Axis:=MoverAxis , 
	Execute:= TRUE, 
	ContinuousUpdate:= TRUE, 
	Position:= rPosition[15], 
	Velocity:= rVelocity [15], 
	Acceleration:= , 
	Deceleration:= , 
	Jerk:= , 
	Gap:= lrCaGap, 
	BufferMode:= , 
	Direction:= , 
	Options:= , 
	Done=> , 
	Busy=> , 
	Active=> , 
	CommandAborted=> , 
	Error=> , 
	ErrorId=> );
	
	IF mcMoveAbsoluteCA.Done AND STATIONDONE[15] THEN
		nMoverSequence :=160;
		STATIONDONE[15]			:=FALSE;
	END_IF
	END_IF
//	TonWait_st[15](IN:=FALSE , PT:=TonWait_PT[15] , Q=> , ET=> );
	
	155:
(*	TonWait_st[15](IN:=TRUE , PT:=TonWait_PT[15] , Q=> , ET=> );
	IF TonWait_st[15].Q THEN
		nMoverSequence :=160;
	END_IF*)
	
	
	160:
	IF POS_BYPASS[16] THEN
	nMoverSequence:=170;
	ELSE  
	mcMoveAbsoluteCA(
	Axis:=MoverAxis , 
	Execute:= FALSE, 
	ContinuousUpdate:= TRUE, 
	Position:= rPosition[16], 
	Velocity:= rVelocity [16], 
	Acceleration:= , 
	Deceleration:= , 
	Jerk:= , 
	Gap:= lrCaGap, 
	BufferMode:= , 
	Direction:= , 
	Options:= , 
	Done=> , 
	Busy=> , 
	Active=> , 
	CommandAborted=> , 
	Error=> , 
	ErrorId=> );
	STATIONDONE[16]			:=FALSE;
	IF STATIONDONE[16]=FALSE THEN
	nMoverSequence :=161;
	END_IF
	END_IF
	
	161:
	IF POS_BYPASS[16] THEN
	nMoverSequence:=170;
	ELSE 
	mcMoveAbsoluteCA(
	Axis:=MoverAxis , 
	Execute:= TRUE, 
	ContinuousUpdate:= TRUE, 
	Position:= rPosition[16], 
	Velocity:= rVelocity [16], 
	Acceleration:= , 
	Deceleration:= , 
	Jerk:= , 
	Gap:= lrCaGap , 
	BufferMode:= , 
	Direction:= , 
	Options:= , 
	Done=> , 
	Busy=> , 
	Active=> , 
	CommandAborted=> , 
	Error=> , 
	ErrorId=> );
	
	IF mcMoveAbsoluteCA.Done AND STATIONDONE[16] THEN
		nMoverSequence :=170;
		STATIONDONE[16]			:=FALSE;
	END_IF
	END_IF
//	TonWait_st[16](IN:=FALSE , PT:=TonWait_PT[16] , Q=> , ET=> );
	
//	165:
(*	TonWait_st[16](IN:=TRUE , PT:=TonWait_PT[16] , Q=> , ET=> );
	IF TonWait_st[16].Q THEN
		nMoverSequence :=170;
	END_IF*)
	
	170:
	IF POS_BYPASS[17] THEN
	nMoverSequence:=180;
	ELSE 
	mcMoveAbsoluteCA(
	Axis:=MoverAxis , 
	Execute:= FALSE, 
	ContinuousUpdate:= TRUE, 
	Position:= rPosition[17], 
	Velocity:= rVelocity [17], 
	Acceleration:= , 
	Deceleration:= , 
	Jerk:= , 
	Gap:=  lrCaGap, 
	BufferMode:= , 
	Direction:= , 
	Options:= , 
	Done=> , 
	Busy=> , 
	Active=> , 
	CommandAborted=> , 
	Error=> , 
	ErrorId=> );
	STATIONDONE[17]			:=FALSE;
	IF STATIONDONE[17]=FALSE THEN
	nMoverSequence :=171;
	END_IF
	END_IF
	
	
	171:
	IF POS_BYPASS[17] THEN
	nMoverSequence:=180;
	ELSE  
	mcMoveAbsoluteCA(
	Axis:=MoverAxis , 
	Execute:= TRUE, 
	ContinuousUpdate:= TRUE, 
	Position:= rPosition[17], 
	Velocity:= rVelocity [17], 
	Acceleration:= , 
	Deceleration:= , 
	Jerk:= , 
	Gap:= lrCaGap, 
	BufferMode:= , 
	Direction:= , 
	Options:= , 
	Done=> , 
	Busy=> , 
	Active=> , 
	CommandAborted=> , 
	Error=> , 
	ErrorId=> );
	
	IF mcMoveAbsoluteCA.Done AND STATIONDONE[17] THEN
		nMoverSequence :=180;
		STATIONDONE[17]			:=FALSE;
	END_IF
	END_IF
//	TonWait_st[17](IN:=FALSE , PT:=TonWait_PT[17] , Q=> , ET=> );
	
//	175:
(*	TonWait_st[17](IN:=TRUE , PT:=TonWait_PT[17] , Q=> , ET=> );
	IF TonWait_st[17].Q THEN
		nMoverSequence :=180;
	END_IF*)

180:
	IF POS_BYPASS[18] THEN
	nMoverSequence:=190;
	ELSE 
	mcMoveAbsoluteCA(
	Axis:=MoverAxis , 
	Execute:= FALSE, 
	ContinuousUpdate:= TRUE, 
	Position:= rPosition[18], 
	Velocity:= rVelocity [18], 
	Acceleration:= , 
	Deceleration:= , 
	Jerk:= , 
	Gap:= lrCaGap, 
	BufferMode:= , 
	Direction:= , 
	Options:= , 
	Done=> , 
	Busy=> , 
	Active=> , 
	CommandAborted=> , 
	Error=> , 
	ErrorId=> );
	STATIONDONE[18]			:=FALSE;
	IF STATIONDONE[18]=FALSE THEN
	nMoverSequence :=181;
	END_IF
	END_IF
	
	
	181:
	IF POS_BYPASS[18] THEN
	nMoverSequence:=190;
	ELSE  
	mcMoveAbsoluteCA(
	Axis:=MoverAxis , 
	Execute:= TRUE, 
	ContinuousUpdate:= TRUE, 
	Position:= rPosition[18], 
	Velocity:= rVelocity [18], 
	Acceleration:= , 
	Deceleration:= , 
	Jerk:= , 
	Gap:= lrCaGap, 
	BufferMode:= , 
	Direction:= , 
	Options:= , 
	Done=> , 
	Busy=> axis_busy, 
	Active=> , 
	CommandAborted=> , 
	Error=> , 
	ErrorId=> );
	
	IF mcMoveAbsoluteCA.Done AND STATIONDONE[18] THEN
		nMoverSequence 				:=190;
		STATIONDONE[18]			:=FALSE;
	END_IF
	END_IF
//	TonWait_st[1](IN:=FALSE , PT:=TonWait_PT[1] , Q=> , ET=> );
//	15:
(*	TonWait_st[1](IN:=TRUE , PT:=TonWait_PT[1] , Q=> , ET=> );
	IF TonWait_st[1].Q THEN
		nMoverSequence :=20;
	END_IF *)
	

	190:
	IF POS_BYPASS[19] THEN
	nMoverSequence:=200;
	ELSE  
	mcMoveAbsoluteCA(
	Axis:=MoverAxis , 
	Execute:= FALSE, 
	ContinuousUpdate:= TRUE, 
	Position:= rPosition[19], 
	Velocity:= rVelocity [19], 
	Acceleration:= , 
	Deceleration:= , 
	Jerk:= , 
	Gap:= lrCaGap , 
	BufferMode:= , 
	Direction:= , 
	Options:= , 
	Done=> , 
	Busy=> , 
	Active=> , 
	CommandAborted=> , 
	Error=> , 
	ErrorId=> );
	STATIONDONE[19]:=FALSE;
	IF STATIONDONE[19]=FALSE THEN
	nMoverSequence :=191;
	END_IF
	END_IF
	
	191:
	IF POS_BYPASS[19] THEN
	nMoverSequence:=200;
	ELSE  
	mcMoveAbsoluteCA(
	Axis:=MoverAxis , 
	Execute:= TRUE, 
	ContinuousUpdate:= TRUE, 
	Position:= rPosition[19], 
	Velocity:= rVelocity [19], 
	Acceleration:= , 
	Deceleration:= , 
	Jerk:= , 
	Gap:= lrCaGap, 
	BufferMode:= , 
	Direction:= , 
	Options:= , 
	Done=> , 
	Busy=> , 
	Active=> , 
	CommandAborted=> , 
	Error=> , 
	ErrorId=> );
	
	IF mcMoveAbsoluteCA.Done AND STATIONDONE[19] THEN
		nMoverSequence :=200;
		STATIONDONE[19]			:=FALSE;
	END_IF
	END_IF
//	TonWait_st[2](IN:=FALSE , PT:=TonWait_PT[2] , Q=> , ET=> );
//	25:
(*	TonWait_st[2](IN:=TRUE , PT:=TonWait_PT[2] , Q=> , ET=> );
	IF TonWait_st[2].Q THEN
		nMoverSequence :=30;
	END_IF *)
	
	

	
	200:
	IF POS_BYPASS[20] THEN
	nMoverSequence:=210;
	ELSE 
	mcMoveAbsoluteCA(
	Axis:=MoverAxis , 
	Execute:= FALSE, 
	ContinuousUpdate:= TRUE, 
	Position:= rPosition[20], 
	Velocity:= rVelocity [20], 
	Acceleration:= , 
	Deceleration:= , 
	Jerk:= , 
	Gap:= lrCaGap, 
	BufferMode:= , 
	Direction:= , 
	Options:= , 
	Done=> , 
	Busy=> , 
	Active=> , 
	CommandAborted=> , 
	Error=> , 
	ErrorId=> );
	STATIONDONE[20]			:=FALSE;
	IF STATIONDONE[20]=FALSE THEN
	nMoverSequence :=201;
	END_IF
	END_IF
	
	201:
	IF POS_BYPASS[20] THEN
	nMoverSequence:=210;
	ELSE  
	mcMoveAbsoluteCA(
	Axis:=MoverAxis , 
	Execute:= TRUE, 
	ContinuousUpdate:= TRUE, 
	Position:= rPosition[20], 
	Velocity:= rVelocity [20], 
	Acceleration:= , 
	Deceleration:= , 
	Jerk:= , 
	Gap:= lrCaGap, 
	BufferMode:= , 
	Direction:= , 
	Options:= , 
	Done=> , 
	Busy=> , 
	Active=> , 
	CommandAborted=> , 
	Error=> , 
	ErrorId=> );
	
	IF mcMoveAbsoluteCA.Done AND STATIONDONE[20] THEN
		nMoverSequence :=210;
		STATIONDONE[20]			:=FALSE;
	END_IF
	END_IF
//	TonWait_st[3](IN:=FALSE , PT:=TonWait_PT[3] , Q=> , ET=> );
	
//	35:
(*	TonWait_st[3](IN:=TRUE , PT:=TonWait_PT[3] , Q=> , ET=> );
	IF TonWait_st[3].Q THEN
		nMoverSequence :=40;
	END_IF*)
	
	
	210:
	IF POS_BYPASS[21] THEN
	nMoverSequence:=220;
	ELSE  
	mcMoveAbsoluteCA(
	Axis:=MoverAxis , 
	Execute:= FALSE, 
	ContinuousUpdate:= TRUE, 
	Position:= rPosition[21], 
	Velocity:= rVelocity [21], 
	Acceleration:= , 
	Deceleration:= , 
	Jerk:= , 
	Gap:= lrCaGap, 
	BufferMode:= , 
	Direction:= , 
	Options:= , 
	Done=> , 
	Busy=> , 
	Active=> , 
	CommandAborted=> , 
	Error=> , 
	ErrorId=> );
	STATIONDONE[21]			:=FALSE;
	IF STATIONDONE[21]=FALSE THEN
	nMoverSequence :=211;
	END_IF
	END_IF
	
	
	211:
	IF POS_BYPASS[21] THEN
	nMoverSequence:=220;
	ELSE  
	mcMoveAbsoluteCA(
	Axis:=MoverAxis , 
	Execute:= TRUE, 
	ContinuousUpdate:= TRUE, 
	Position:= rPosition[21], 
	Velocity:= rVelocity [21], 
	Acceleration:= , 
	Deceleration:= , 
	Jerk:= , 
	Gap:= lrCaGap , 
	BufferMode:= , 
	Direction:= , 
	Options:= , 
	Done=> , 
	Busy=> , 
	Active=> , 
	CommandAborted=> , 
	Error=> , 
	ErrorId=> );
	
	IF mcMoveAbsoluteCA.Done AND STATIONDONE[21] THEN
		nMoverSequence :=220;
		STATIONDONE[21]			:=FALSE;
	END_IF
	END_IF
//	TonWait_st[4](IN:=FALSE , PT:=TonWait_PT[4] , Q=> , ET=> );
	
//	45:
(*	TonWait_st[4](IN:=TRUE , PT:=TonWait_PT[4] , Q=> , ET=> );
	IF TonWait_st[4].Q THEN
		nMoverSequence :=50;
	END_IF*)
	
	
	220:
	IF POS_BYPASS[22] THEN
	nMoverSequence:=230;
	ELSE  
	mcMoveAbsoluteCA(
	Axis:=MoverAxis , 
	Execute:= FALSE, 
	ContinuousUpdate:= TRUE, 
	Position:= rPosition[22], 
	Velocity:= rVelocity [22], 
	Acceleration:= , 
	Deceleration:= , 
	Jerk:= , 
	Gap:= lrCaGap , 
	BufferMode:= , 
	Direction:= , 
	Options:= , 
	Done=> , 
	Busy=> , 
	Active=> , 
	CommandAborted=> , 
	Error=> , 
	ErrorId=> );
	STATIONDONE[22]			:=FALSE;
	IF STATIONDONE[22]=FALSE THEN
	nMoverSequence :=221;
	END_IF
	END_IF
	
	
	221:
	IF POS_BYPASS[22] THEN
	nMoverSequence:=230;
	ELSE 
	mcMoveAbsoluteCA(
	Axis:=MoverAxis , 
	Execute:= TRUE, 
	ContinuousUpdate:= TRUE, 
	Position:= rPosition[22], 
	Velocity:= rVelocity [22], 
	Acceleration:= , 
	Deceleration:= , 
	Jerk:= , 
	Gap:= lrCaGap, 
	BufferMode:= , 
	Direction:= , 
	Options:= , 
	Done=> , 
	Busy=> , 
	Active=> , 
	CommandAborted=> , 
	Error=> , 
	ErrorId=> );
	
	IF mcMoveAbsoluteCA.Done AND STATIONDONE[22] THEN
		nMoverSequence :=230;
		STATIONDONE[22]			:=FALSE;
	END_IF
	END_IF
//	TonWait_st[5](IN:=FALSE , PT:=TonWait_PT[5] , Q=> , ET=> );
	
//	55:
(*	TonWait_st[5](IN:=TRUE , PT:=TonWait_PT[5] , Q=> , ET=> );
	IF TonWait_st[5].Q THEN
		nMoverSequence :=60;
	END_IF*)
	
	
	230:
	IF POS_BYPASS[23] THEN
	nMoverSequence:=240;
	ELSE  
	mcMoveAbsoluteCA(
	Axis:=MoverAxis , 
	Execute:= FALSE, 
	ContinuousUpdate:= TRUE, 
	Position:= rPosition[23], 
	Velocity:= rVelocity [23], 
	Acceleration:= , 
	Deceleration:= , 
	Jerk:= , 
	Gap:= lrCaGap , 
	BufferMode:= , 
	Direction:= , 
	Options:= , 
	Done=> , 
	Busy=> , 
	Active=> , 
	CommandAborted=> , 
	Error=> , 
	ErrorId=> );
	STATIONDONE[23]			:=FALSE;
	IF STATIONDONE[23]=FALSE THEN
	nMoverSequence :=231;
	END_IF
	END_IF
	
	231:
	IF POS_BYPASS[23] THEN
	nMoverSequence:=240;
	ELSE   
	mcMoveAbsoluteCA(
	Axis:=MoverAxis , 
	Execute:= TRUE, 
	ContinuousUpdate:= TRUE, 
	Position:= rPosition[23], 
	Velocity:= rVelocity [23], 
	Acceleration:= , 
	Deceleration:= , 
	Jerk:= , 
	Gap:= lrCaGap , 
	BufferMode:= , 
	Direction:= , 
	Options:= , 
	Done=> , 
	Busy=> , 
	Active=> , 
	CommandAborted=> , 
	Error=> , 
	ErrorId=> );
	
	IF mcMoveAbsoluteCA.Done AND STATIONDONE[23] THEN
		nMoverSequence :=240;
		STATIONDONE[23]			:=FALSE;
	END_IF
	END_IF
//	TonWait_st[6](IN:=FALSE , PT:=TonWait_PT[6] , Q=> , ET=> );
	
(*	65:
	TonWait_st[6](IN:=TRUE , PT:=TonWait_PT[6] , Q=> , ET=> );
	IF TonWait_st[6].Q THEN
		nMoverSequence :=70;
	END_IF*)
	
	
	240:
	IF POS_BYPASS[24] THEN
	nMoverSequence:=250;
	ELSE  
	mcMoveAbsoluteCA(
	Axis:=MoverAxis , 
	Execute:= FALSE, 
	ContinuousUpdate:= TRUE, 
	Position:= rPosition[24], 
	Velocity:= rVelocity [24], 
	Acceleration:= , 
	Deceleration:= , 
	Jerk:= , 
	Gap:= lrCaGap , 
	BufferMode:= , 
	Direction:= , 
	Options:= , 
	Done=> , 
	Busy=> , 
	Active=> , 
	CommandAborted=> , 
	Error=> , 
	ErrorId=> );
	STATIONDONE[24]			:=FALSE;
	IF STATIONDONE[24]=FALSE THEN
	nMoverSequence :=241;
	END_IF
	END_IF
	
	241:
	IF POS_BYPASS[24] THEN
	nMoverSequence:=250;
	ELSE 
	mcMoveAbsoluteCA(
	Axis:=MoverAxis , 
	Execute:= TRUE, 
	ContinuousUpdate:= TRUE, 
	Position:= rPosition[24], 
	Velocity:= rVelocity [24], 
	Acceleration:= , 
	Deceleration:= , 
	Jerk:= , 
	Gap:= lrCaGap , 
	BufferMode:= , 
	Direction:= , 
	Options:= , 
	Done=> , 
	Busy=> , 
	Active=> , 
	CommandAborted=> , 
	Error=> , 
	ErrorId=> );
	
	IF mcMoveAbsoluteCA.Done AND STATIONDONE[24] THEN
		nMoverSequence :=250;
		STATIONDONE[24]			:=FALSE;
	END_IF
	END_IF
//	TonWait_st[7](IN:=FALSE , PT:=TonWait_PT[7] , Q=> , ET=> );
	
(*	75:
	TonWait_st[7](IN:=TRUE , PT:=TonWait_PT[7] , Q=> , ET=> );
	IF TonWait_st[7].Q THEN
		nMoverSequence :=80;
	END_IF*)
	
	
	250:
	IF POS_BYPASS[25] THEN
	nMoverSequence:=260;
	ELSE 
	mcMoveAbsoluteCA(
	Axis:=MoverAxis , 
	Execute:= FALSE, 
	ContinuousUpdate:= TRUE, 
	Position:= rPosition[25], 
	Velocity:= rVelocity [25], 
	Acceleration:= , 
	Deceleration:= , 
	Jerk:= , 
	Gap:= lrCaGap , 
	BufferMode:= , 
	Direction:= , 
	Options:= , 
	Done=> , 
	Busy=> , 
	Active=> , 
	CommandAborted=> , 
	Error=> , 
	ErrorId=> );
	STATIONDONE[25]			:=FALSE;
	IF STATIONDONE[25]=FALSE THEN
	nMoverSequence :=251;
	END_IF
	END_IF
	
	251:
	IF POS_BYPASS[25] THEN
	nMoverSequence:=260;
	ELSE 
	mcMoveAbsoluteCA(
	Axis:=MoverAxis , 
	Execute:= TRUE, 
	ContinuousUpdate:= TRUE, 
	Position:= rPosition[25], 
	Velocity:= rVelocity [25], 
	Acceleration:= , 
	Deceleration:= , 
	Jerk:= , 
	Gap:= lrCaGap, 
	BufferMode:= , 
	Direction:= , 
	Options:= , 
	Done=> , 
	Busy=> , 
	Active=> , 
	CommandAborted=> , 
	Error=> , 
	ErrorId=> );
	
	IF mcMoveAbsoluteCA.Done AND STATIONDONE[25] THEN
		nMoverSequence :=260;
		STATIONDONE[25]			:=FALSE;
	END_IF
	END_IF
//	TonWait_st[8](IN:=FALSE , PT:=TonWait_PT[8] , Q=> , ET=> );
	
(*	85:
	TonWait_st[8](IN:=TRUE , PT:=TonWait_PT[8] , Q=> , ET=> );
	IF TonWait_st[8].Q THEN
		nMoverSequence :=90;
	END_IF*)
	
	
	260:
	IF POS_BYPASS[26] THEN
	nMoverSequence:=270;
	ELSE 
	mcMoveAbsoluteCA(
	Axis:=MoverAxis , 
	Execute:= FALSE, 
	ContinuousUpdate:= TRUE, 
	Position:= rPosition[26], 
	Velocity:= rVelocity [26], 
	Acceleration:= , 
	Deceleration:= , 
	Jerk:= , 
	Gap:= lrCaGap , 
	BufferMode:= , 
	Direction:= , 
	Options:= , 
	Done=> , 
	Busy=> , 
	Active=> , 
	CommandAborted=> , 
	Error=> , 
	ErrorId=> );
	STATIONDONE[26]			:=FALSE;
	IF STATIONDONE[26]=FALSE THEN
	nMoverSequence :=261;
	END_IF
	END_IF
	
	
	261:
	IF POS_BYPASS[26] THEN
	nMoverSequence:=270;
	ELSE 
	mcMoveAbsoluteCA(
	Axis:=MoverAxis , 
	Execute:= TRUE, 
	ContinuousUpdate:= TRUE, 
	Position:= rPosition[26], 
	Velocity:= rVelocity [26], 
	Acceleration:= , 
	Deceleration:= , 
	Jerk:= , 
	Gap:= lrCaGap , 
	BufferMode:= , 
	Direction:= , 
	Options:= , 
	Done=> , 
	Busy=> , 
	Active=> , 
	CommandAborted=> , 
	Error=> , 
	ErrorId=> );
	
	IF mcMoveAbsoluteCA.Done AND STATIONDONE[26] THEN
		nMoverSequence :=270;
		STATIONDONE[26]			:=FALSE;
	END_IF
	END_IF
//	TonWait_st[9](IN:=FALSE , PT:=TonWait_PT[9] , Q=> , ET=> );
	
(*	95:
	TonWait_st[9](IN:=TRUE , PT:=TonWait_PT[9] , Q=> , ET=> );
	IF TonWait_st[9].Q THEN
		nMoverSequence :=100;
	END_IF *)
	
	
	270:
	IF POS_BYPASS[27] THEN
	nMoverSequence:=280;
	ELSE 
	mcMoveAbsoluteCA(
	Axis:=MoverAxis , 
	Execute:= FALSE, 
	ContinuousUpdate:= TRUE, 
	Position:= rPosition[27], 
	Velocity:= rVelocity [27], 
	Acceleration:= , 
	Deceleration:= , 
	Jerk:= , 
	Gap:= lrCaGap, 
	BufferMode:= , 
	Direction:= , 
	Options:= , 
	Done=> , 
	Busy=> , 
	Active=> , 
	CommandAborted=> , 
	Error=> , 
	ErrorId=> );
	STATIONDONE[27]			:=FALSE;
	IF STATIONDONE[27]=FALSE THEN
	nMoverSequence :=271;
	END_IF
	END_IF
	
	271:
	IF POS_BYPASS[27] THEN
	nMoverSequence:=280;
	ELSE  
	mcMoveAbsoluteCA(
	Axis:=MoverAxis , 
	Execute:= TRUE, 
	ContinuousUpdate:= TRUE, 
	Position:= rPosition[27], 
	Velocity:= rVelocity [27], 
	Acceleration:= , 
	Deceleration:= , 
	Jerk:= , 
	Gap:= lrCaGap , 
	BufferMode:= , 
	Direction:= , 
	Options:= , 
	Done=> , 
	Busy=> , 
	Active=> , 
	CommandAborted=> , 
	Error=> , 
	ErrorId=> );
	
	IF mcMoveAbsoluteCA.Done AND STATIONDONE[27] THEN
		nMoverSequence :=280;
		STATIONDONE[27]			:=FALSE;
	END_IF
	END_IF
//	TonWait_st[10](IN:=FALSE , PT:=TonWait_PT[10] , Q=> , ET=> );
	
(*	105:
	TonWait_st[10](IN:=TRUE , PT:=TonWait_PT[10] , Q=> , ET=> );
	IF TonWait_st[10].Q THEN
		nMoverSequence :=110;
	END_IF*)
	
	
	280:
	IF POS_BYPASS[28] THEN
	nMoverSequence:=290;
	ELSE  
	mcMoveAbsoluteCA(
	Axis:=MoverAxis , 
	Execute:= FALSE, 
	ContinuousUpdate:= TRUE, 
	Position:= rPosition[28], 
	Velocity:= rVelocity [28], 
	Acceleration:= , 
	Deceleration:= , 
	Jerk:= , 
	Gap:= lrCaGap , 
	BufferMode:= , 
	Direction:= , 
	Options:= , 
	Done=> , 
	Busy=> , 
	Active=> , 
	CommandAborted=> , 
	Error=> , 
	ErrorId=> );
	STATIONDONE[28]			:=FALSE;
	IF STATIONDONE[28]=FALSE THEN
	nMoverSequence :=281;
	END_IF
	END_IF
	
	281:
	IF POS_BYPASS[28] THEN
	nMoverSequence:=290;
	ELSE 
	mcMoveAbsoluteCA(
	Axis:=MoverAxis , 
	Execute:= TRUE, 
	ContinuousUpdate:= TRUE, 
	Position:= rPosition[28], 
	Velocity:= rVelocity [28], 
	Acceleration:= , 
	Deceleration:= , 
	Jerk:= , 
	Gap:= lrCaGap, 
	BufferMode:= , 
	Direction:= , 
	Options:= , 
	Done=> , 
	Busy=> , 
	Active=> , 
	CommandAborted=> , 
	Error=> , 
	ErrorId=> );
	
	IF mcMoveAbsoluteCA.Done AND STATIONDONE[28] THEN
		nMoverSequence :=290;
		STATIONDONE[28]			:=FALSE;
	END_IF
	END_IF
//	TonWait_st[11](IN:=FALSE , PT:=TonWait_PT[11] , Q=> , ET=> );
	
(*	115:
	TonWait_st[11](IN:=TRUE , PT:=TonWait_PT[11] , Q=> , ET=> );
	IF TonWait_st[11].Q THEN
		nMoverSequence :=120;
	END_IF*)
	
	
	290:
	IF POS_BYPASS[29] THEN
	nMoverSequence:=300;
	ELSE 
	mcMoveAbsoluteCA(
	Axis:=MoverAxis , 
	Execute:= FALSE, 
	ContinuousUpdate:= TRUE, 
	Position:= rPosition[29], 
	Velocity:= rVelocity [29], 
	Acceleration:= , 
	Deceleration:= , 
	Jerk:= , 
	Gap:= lrCaGap , 
	BufferMode:= , 
	Direction:= , 
	Options:= , 
	Done=> , 
	Busy=> , 
	Active=> , 
	CommandAborted=> , 
	Error=> , 
	ErrorId=> );
	STATIONDONE[29]	:=FALSE;
	IF STATIONDONE[29]=FALSE THEN
	nMoverSequence :=291;
	END_IF
	END_IF
	
	
	291:
	IF POS_BYPASS[29] THEN
	nMoverSequence:=300;
	ELSE 
	mcMoveAbsoluteCA(
	Axis:=MoverAxis , 
	Execute:= TRUE, 
	ContinuousUpdate:= TRUE, 
	Position:= rPosition[29], 
	Velocity:= rVelocity [29], 
	Acceleration:= , 
	Deceleration:= , 
	Jerk:= , 
	Gap:= lrCaGap, 
	BufferMode:= , 
	Direction:= , 
	Options:= , 
	Done=> , 
	Busy=> , 
	Active=> , 
	CommandAborted=> , 
	Error=> , 
	ErrorId=> );
	
	IF mcMoveAbsoluteCA.Done AND STATIONDONE[29] THEN
		nMoverSequence :=300;
		STATIONDONE[29]			:=FALSE;
	END_IF
	END_IF
//	TonWait_st[12](IN:=FALSE , PT:=TonWait_PT[12] , Q=> , ET=> );
	
(*	125:
	TonWait_st[12](IN:=TRUE , PT:=TonWait_PT[12] , Q=> , ET=> );
	IF TonWait_st[12].Q THEN
		nMoverSequence :=130;
	END_IF*)
	
	300:
	IF POS_BYPASS[30] THEN
	nMoverSequence:=310;
	ELSE  
	mcMoveAbsoluteCA(
	Axis:=MoverAxis , 
	Execute:= FALSE, 
	ContinuousUpdate:= TRUE, 
	Position:= rPosition[30], 
	Velocity:= rVelocity [30], 
	Acceleration:= , 
	Deceleration:= , 
	Jerk:= , 
	Gap:= lrCaGap, 
	BufferMode:= , 
	Direction:= , 
	Options:= , 
	Done=> , 
	Busy=> , 
	Active=> , 
	CommandAborted=> , 
	Error=> , 
	ErrorId=> );
	STATIONDONE[30]			:=FALSE;
	IF STATIONDONE[30]=FALSE THEN
	nMoverSequence :=301;
	END_IF
	END_IF
	
	301:
	IF POS_BYPASS[30] THEN
	nMoverSequence:=310;
	ELSE 
	mcMoveAbsoluteCA(
	Axis:=MoverAxis , 
	Execute:= TRUE, 
	ContinuousUpdate:= TRUE, 
	Position:= rPosition[30], 
	Velocity:= rVelocity [30], 
	Acceleration:= , 
	Deceleration:= , 
	Jerk:= , 
	Gap:= lrCaGap , 
	BufferMode:= , 
	Direction:= , 
	Options:= , 
	Done=> , 
	Busy=> , 
	Active=> , 
	CommandAborted=> , 
	Error=> , 
	ErrorId=> );
	
	IF mcMoveAbsoluteCA.Done AND STATIONDONE[30] THEN
		nMoverSequence :=310;
		STATIONDONE[30]			:=FALSE;
	END_IF
	END_IF
//	TonWait_st[13](IN:=FALSE , PT:=TonWait_PT[13] , Q=> , ET=> );
	
(*	135:
	TonWait_st[13](IN:=TRUE , PT:=TonWait_PT[13] , Q=> , ET=> );
	IF TonWait_st[13].Q THEN
		nMoverSequence :=140;
	END_IF*)
	
	
	310:
	IF POS_BYPASS[31] THEN
	nMoverSequence:=320;
	ELSE 
	mcMoveAbsoluteCA(
	Axis:=MoverAxis , 
	Execute:= FALSE, 
	ContinuousUpdate:= TRUE, 
	Position:= rPosition[31], 
	Velocity:= rVelocity [31], 
	Acceleration:= , 
	Deceleration:= , 
	Jerk:= , 
	Gap:= lrCaGap, 
	BufferMode:= , 
	Direction:= , 
	Options:= , 
	Done=> , 
	Busy=> , 
	Active=> , 
	CommandAborted=> , 
	Error=> , 
	ErrorId=> );
	STATIONDONE[31]			:=FALSE;
	IF STATIONDONE[31]=FALSE THEN
	nMoverSequence :=311;
	END_IF
	END_IF
	
	
	311:
	IF POS_BYPASS[31] THEN
	nMoverSequence:=320;
	ELSE  
	mcMoveAbsoluteCA(
	Axis:=MoverAxis , 
	Execute:= TRUE, 
	ContinuousUpdate:= TRUE, 
	Position:= rPosition[31], 
	Velocity:= rVelocity [31], 
	Acceleration:= , 
	Deceleration:= , 
	Jerk:= , 
	Gap:= lrCaGap, 
	BufferMode:= , 
	Direction:= , 
	Options:= , 
	Done=> , 
	Busy=> , 
	Active=> , 
	CommandAborted=> , 
	Error=> , 
	ErrorId=> );
	
	IF mcMoveAbsoluteCA.Done AND STATIONDONE[31] THEN
		nMoverSequence :=320;
		STATIONDONE[31]			:=FALSE;
	END_IF
	END_IF
//	TonWait_st[14](IN:=FALSE , PT:=TonWait_PT[14] , Q=> , ET=> );
	
(*	145:
	TonWait_st[14](IN:=TRUE , PT:=TonWait_PT[14] , Q=> , ET=> );
	IF TonWait_st[14].Q THEN
		nMoverSequence :=150;
	END_IF*)
	
	
	320:
	IF POS_BYPASS[32] THEN
	nMoverSequence:=330;
	ELSE 
	mcMoveAbsoluteCA(
	Axis:=MoverAxis , 
	Execute:= FALSE, 
	ContinuousUpdate:= TRUE, 
	Position:= rPosition[32], 
	Velocity:= rVelocity [32], 
	Acceleration:= , 
	Deceleration:= , 
	Jerk:= , 
	Gap:= lrCaGap, 
	BufferMode:= , 
	Direction:= , 
	Options:= , 
	Done=> , 
	Busy=> , 
	Active=> , 
	CommandAborted=> , 
	Error=> , 
	ErrorId=> );
	STATIONDONE[32]			:=FALSE;
	IF STATIONDONE[32]=FALSE THEN
	nMoverSequence :=321;
	END_IF
	END_IF
	
	321:
	IF POS_BYPASS[32] THEN
	nMoverSequence:=330;
	ELSE  
	mcMoveAbsoluteCA(
	Axis:=MoverAxis , 
	Execute:= TRUE, 
	ContinuousUpdate:= TRUE, 
	Position:= rPosition[32], 
	Velocity:= rVelocity [32], 
	Acceleration:= , 
	Deceleration:= , 
	Jerk:= , 
	Gap:= lrCaGap, 
	BufferMode:= , 
	Direction:= , 
	Options:= , 
	Done=> , 
	Busy=> , 
	Active=> , 
	CommandAborted=> , 
	Error=> , 
	ErrorId=> );
	
	IF mcMoveAbsoluteCA.Done AND STATIONDONE[32] THEN
		nMoverSequence :=330;
		STATIONDONE[32]			:=FALSE;
	END_IF
	END_IF
//	TonWait_st[15](IN:=FALSE , PT:=TonWait_PT[15] , Q=> , ET=> );
	
(*	155:
	TonWait_st[15](IN:=TRUE , PT:=TonWait_PT[15] , Q=> , ET=> );
	IF TonWait_st[15].Q THEN
		nMoverSequence :=160;
	END_IF*)
	
	
	330:
	IF POS_BYPASS[33] THEN
	nMoverSequence:=340;
	ELSE  
	mcMoveAbsoluteCA(
	Axis:=MoverAxis , 
	Execute:= FALSE, 
	ContinuousUpdate:= TRUE, 
	Position:= rPosition[33], 
	Velocity:= rVelocity [33], 
	Acceleration:= , 
	Deceleration:= , 
	Jerk:= , 
	Gap:= lrCaGap, 
	BufferMode:= , 
	Direction:= , 
	Options:= , 
	Done=> , 
	Busy=> , 
	Active=> , 
	CommandAborted=> , 
	Error=> , 
	ErrorId=> );
	STATIONDONE[33]			:=FALSE;
	IF STATIONDONE[33]=FALSE THEN
	nMoverSequence :=331;
	END_IF
	END_IF
	
	
	331:
	IF POS_BYPASS[33] THEN
	nMoverSequence:=340;
	ELSE 
	mcMoveAbsoluteCA(
	Axis:=MoverAxis , 
	Execute:= TRUE, 
	ContinuousUpdate:= TRUE, 
	Position:= rPosition[33], 
	Velocity:= rVelocity [33], 
	Acceleration:= , 
	Deceleration:= , 
	Jerk:= , 
	Gap:= lrCaGap , 
	BufferMode:= , 
	Direction:= , 
	Options:= , 
	Done=> , 
	Busy=> , 
	Active=> , 
	CommandAborted=> , 
	Error=> , 
	ErrorId=> );
	
	IF mcMoveAbsoluteCA.Done AND STATIONDONE[33] THEN
		nMoverSequence :=340;
		STATIONDONE[33]			:=FALSE;
	END_IF
	END_IF
//	TonWait_st[16](IN:=FALSE , PT:=TonWait_PT[16] , Q=> , ET=> );
	
(*	165:
	TonWait_st[16](IN:=TRUE , PT:=TonWait_PT[16] , Q=> , ET=> );
	IF TonWait_st[16].Q THEN
		nMoverSequence :=170;
	END_IF*)
	
	340:
	IF POS_BYPASS[34] THEN
	nMoverSequence:=350;
	ELSE
	mcMoveAbsoluteCA(
	Axis:=MoverAxis , 
	Execute:= FALSE, 
	ContinuousUpdate:= TRUE, 
	Position:= rPosition[34], 
	Velocity:= rVelocity [34], 
	Acceleration:= , 
	Deceleration:= , 
	Jerk:= , 
	Gap:=  lrCaGap, 
	BufferMode:= , 
	Direction:= , 
	Options:= , 
	Done=> , 
	Busy=> , 
	Active=> , 
	CommandAborted=> , 
	Error=> , 
	ErrorId=> );
	STATIONDONE[34]			:=FALSE;
	IF STATIONDONE[34]=FALSE THEN
	nMoverSequence :=341;
	END_IF
	END_IF
	
	341:
	IF POS_BYPASS[34] THEN
	nMoverSequence:=350;
	ELSE 
	mcMoveAbsoluteCA(
	Axis:=MoverAxis , 
	Execute:= TRUE, 
	ContinuousUpdate:= TRUE, 
	Position:= rPosition[34], 
	Velocity:= rVelocity [34], 
	Acceleration:= , 
	Deceleration:= , 
	Jerk:= , 
	Gap:= lrCaGap, 
	BufferMode:= , 
	Direction:= , 
	Options:= , 
	Done=> , 
	Busy=> , 
	Active=> , 
	CommandAborted=> , 
	Error=> , 
	ErrorId=> );
	
	IF mcMoveAbsoluteCA.Done AND STATIONDONE[34] THEN
		nMoverSequence :=350;
		STATIONDONE[34]			:=FALSE;
	END_IF
	END_IF
//	TonWait_st[17](IN:=FALSE , PT:=TonWait_PT[17] , Q=> , ET=> );
	
(*	175:
	TonWait_st[17](IN:=TRUE , PT:=TonWait_PT[17] , Q=> , ET=> );
	IF TonWait_st[17].Q THEN
		nMoverSequence :=180;
	END_IF*)

	350:
	IF POS_BYPASS[35] THEN
	nMoverSequence:=360;
	ELSE 
	mcMoveAbsoluteCA(
	Axis:=MoverAxis , 
	Execute:= FALSE, 
	ContinuousUpdate:= TRUE, 
	Position:= rPosition[35], 
	Velocity:= rVelocity [35], 
	Acceleration:= , 
	Deceleration:= , 
	Jerk:= , 
	Gap:=  lrCaGap, 
	BufferMode:= , 
	Direction:= , 
	Options:= , 
	Done=> , 
	Busy=> , 
	Active=> , 
	CommandAborted=> , 
	Error=> , 
	ErrorId=> );
	STATIONDONE[35]					:=FALSE;
	IF STATIONDONE[35]=FALSE THEN
	nMoverSequence :=351;
	END_IF
	END_IF
	
	351:
	IF POS_BYPASS[35] THEN
	nMoverSequence:=360;
	ELSE 
	mcMoveAbsoluteCA(
	Axis:=MoverAxis , 
	Execute:= TRUE, 
	ContinuousUpdate:= TRUE, 
	Position:= rPosition[35], 
	Velocity:= rVelocity [35], 
	Acceleration:= , 
	Deceleration:= , 
	Jerk:= , 
	Gap:= lrCaGap, 
	BufferMode:= , 
	Direction:= , 
	Options:= , 
	Done=> , 
	Busy=> , 
	Active=> , 
	CommandAborted=> , 
	Error=> , 
	ErrorId=> );
	
	IF mcMoveAbsoluteCA.Done AND STATIONDONE[35] THEN
		nMoverSequence :=360;
		STATIONDONE[35]					:=FALSE;
	END_IF
	END_IF
//	TonWait_st[17](IN:=FALSE , PT:=TonWait_PT[17] , Q=> , ET=> );
	
(*	175:
	TonWait_st[17](IN:=TRUE , PT:=TonWait_PT[17] , Q=> , ET=> );
	IF TonWait_st[17].Q THEN
		nMoverSequence :=180;
	END_IF*)	
	
	360:
	IF bStopCommandTriggered THEN
		nMoverSequence :=0;
		 bStopCommandTriggered :=FALSE;
		 ELSE
		  nMoverSequence :=10; 
	END_IF
	
	
END_CASE
ELSE
	mc_moverhalt(
	Axis:= MoverAxis, 
	Execute:= TRUE , 
	Deceleration:= , 
	Jerk:= , 
	Gap:= , 
	Options:= , 
	Done=> , 
	Busy=> , 
	Active=> , 
	CommandAborted=> , 
	Error=> , 
	ErrorId=> );
	
	
	mcMoveAbsoluteCA(
	Axis:=MoverAxis , 
	Execute:= FALSE, 
	ContinuousUpdate:= TRUE, 
	Position:= , 
	Velocity:= , 
	Acceleration:= , 
	Deceleration:= , 
	Jerk:= , 
	Gap:= lrCaGap, 
	BufferMode:= , 
	Direction:= , 
	Options:= , 
	Done=> , 
	Busy=> , 
	Active=> , 
	CommandAborted=> , 
	Error=> , 
	ErrorId=> );
	nMoverSequence := nMoverSequence;
	
END_IF

IF R_TRIG_Run.Q THEN
		bStopCommandTriggered :=FALSE;
END_IF
	
POSITION_DONE:=mcMoveAbsoluteCA.Done;

//Test
bStopCommandTriggered := TRUE;
bStopCommandTriggered := TRUE;
bStopCommandTriggered := TRUE;
POSITION_DONE:=mcMoveAbsoluteCA.Done;

END_FUNCTION_BLOCK

// ---- POUs/GENERAL/EtherCatDiag.TcPOU
PROGRAM EtherCatDiag
VAR
	bena: BOOL;
	test : Tc2_Standard.R_TRIG;
	
	(* Execute *)
	bExecute_X1: 					BOOL;
	
	(* FB's Required *)
	fbGetCfgSlaves_X1  			: FB_EcGetConfSlaves;       //Get Slave Details
	fbGetAllSlaveStates_X1			: FB_EcGetAllSlaveStates;   //Get Slave State
	
	(* Status *)
	nCfgSlaveCount_X1				: UINT;                     //Actual Slave Count (Slave Details)
	nEcSlavesRead_X1				: UINT;						//Actual Salve Count (Slave State)
	
	(* POU Var *)
	sEcMasterNetId_X1			: T_AmsNetId;               //Ams NetID X1
	ArrEcConfSlaveInfo_X1: ARRAY [1..GVL.ECAT_MAX_SLAVES_X1] OF ST_EcSlaveConfigData; //Slave Details Array
	ArrEcSlaveState_X1:	ARRAY [1..GVL.ECAT_MAX_SLAVES_X1] OF ST_EcSlaveState;		//Slave State Array
	I_X1: INT;
	iDiagIndex_X1					: ARRAY [0..3] OF UINT;
	sState_X1: STRING;
	arrSlaveInfo_X1 				: ARRAY [1..GVL.ECAT_MAX_SLAVES_X1] OF ST_SlaveStateInfo; //Slave Data
	
	(* Error Count *)
	bCheckError : BOOL;
	nNodeErrorCount   : INT;
	N_X1:INT:=1;
	ErrorState_X1:INT;
	fbGetSlaveState_X1     : FB_EcReqSlaveState;
	
END_VAR

test(CLK:=bena,Q=>bExecute_X1);

(*Generate NetId*)
sEcMasterNetId_X1 := F_CreateAmsNetId(nIds := GVL.EC_MasterNetID_Arr_X1);

(* Get Configured Slaves *)
fbGetCfgSlaves_X1(
	sNetId:= sEcMasterNetId_X1,
	pArrEcConfSlaveInfo:= ADR(ArrEcConfSlaveInfo_X1),
	cbBufLen:= SIZEOF(ArrEcConfSlaveInfo_X1),
	bExecute	:= bExecute_X1,
	tTimeout:= DEFAULT_ADS_TIMEOUT,
	nSlaves=> nCfgSlaveCount_X1 );

(*Get Slave States*)
fbGetAllSlaveStates_X1(
	sNetId		:= sEcMasterNetId_X1,
	pStateBuf	:= ADR(ArrEcSlaveState_X1),
	cbBufLen	:= SIZEOF(ArrEcSlaveState_X1),
	bExecute	:= bExecute_X1,
	tTimeout	:= DEFAULT_ADS_TIMEOUT,
	nSlaves	=> nEcSlavesRead_X1
);


IF NOT fbGetAllSlaveStates_X1.bBusy THEN
		fbGetCfgSlaves_X1(bExecute:= FALSE);
		fbGetAllSlaveStates_X1(bExecute:= FALSE);
		IF NOT fbGetAllSlaveStates_X1.bError THEN
			IF nEcSlavesRead_X1 = nCfgSlaveCount_X1 THEN
				FOR I_X1 := 0 TO 3 DO
					iDiagIndex_X1[I_X1] := 0;
				END_FOR

